    |   movel([0.123619, -1.308505, -2.621717, -0.782167, 1.570796, 1.694415],accel_mss,speed_ms,0,blend_radius_m)
    |   movel([0.123541, -1.308897, -2.621479, -0.782012, 1.570796, 1.694337],accel_mss,speed_ms,0,blend_radius_m)
    |   movel([0.123274, -1.309201, -2.621295, -0.781893, 1.570796, 1.694070],accel_mss,speed_ms,0,blend_radius_m)
    |   movel([0.122788, -1.309523, -2.621100, -0.781766, 1.570796, 1.693584],accel_mss,speed_ms,0,blend_radius_m)
    |   movel([0.122358, -1.309528, -2.621097, -0.781764, 1.570796, 1.693155],accel_mss,speed_ms,0,blend_radius_m)
    |   movel([0.122204, -1.309206, -2.621292, -0.781891, 1.570796, 1.693000],accel_mss,speed_ms,0,blend_radius_m)
    |   movel([0.122399, -1.308718, -2.621588, -0.782083, 1.570796, 1.693196],accel_mss,speed_ms,0,blend_radius_m)
    |   speed_ms = 0.003
    |   movel([0.122399, -1.294954, -2.615092, -0.802344, 1.570796, 1.693196],accel_mss,speed_ms,0,blend_radius_m)
    |   speed_ms = 1.000
    |   movel([0.122399, -1.268722, -2.601712, -0.841955, 1.570796, 1.693196],accel_mss,speed_ms,0,blend_radius_m)
    |   movel([0.122299, -1.268148, -2.602040, -0.842201, 1.570796, 1.693095],accel_mss,speed_ms,0,blend_radius_m)
    |   movel([0.122299, -1.294388, -2.615427, -0.802573, 1.570796, 1.693095],accel_mss,speed_ms,0,blend_radius_m)
    |   speed_ms = 0.003
    |   movel([0.122299, -1.304675, -2.620314, -0.787400, 1.570796, 1.693095],accel_mss,speed_ms,0,blend_radius_m)
    |   speed_ms = 0.007
    |   movel([0.123492, -1.303784, -2.620850, -0.787755, 1.570796, 1.694289],accel_mss,speed_ms,0,blend_radius_m)
    |   movel([0.124884, -1.303405, -2.621078, -0.787906, 1.570796, 1.695680],accel_mss,speed_ms,0,blend_radius_m)
    |   movel([0.125943, -1.303780, -2.620852, -0.787756, 1.570796, 1.696740],accel_mss,speed_ms,0,blend_radius_m)
    |   movel([0.126327, -1.304786, -2.620247, -0.787356, 1.570796, 1.697123],accel_mss,speed_ms,0,blend_radius_m)
    |   movel([0.125902, -1.306088, -2.619462, -0.786839, 1.570796, 1.696698],accel_mss,speed_ms,0,blend_radius_m)
    |   movel([0.125601, -1.306535, -2.619192, -0.786662, 1.570796, 1.696398],accel_mss,speed_ms,0,blend_radius_m)
    |   movel([0.125298, -1.306889, -2.618978, -0.786522, 1.570796, 1.696095],accel_mss,speed_ms,0,blend_radius_m)
    |   movel([0.124939, -1.307203, -2.618788, -0.786398, 1.570796, 1.695735],accel_mss,speed_ms,0,blend_radius_m)
    |   movel([0.124479, -1.307524, -2.618594, -0.786271, 1.570796, 1.695275],accel_mss,speed_ms,0,blend_radius_m)
    |   movel([0.123696, -1.307924, -2.618351, -0.786113, 1.570796, 1.694492],accel_mss,speed_ms,0,blend_radius_m)
    |   movel([0.122962, -1.308104, -2.618242, -0.786043, 1.570796, 1.693758],accel_mss,speed_ms,0,blend_radius_m)
    |   movel([0.122312, -1.308051, -2.618275, -0.786064, 1.570796, 1.693109],accel_mss,speed_ms,0,blend_radius_m)
    |   movel([0.121777, -1.307771, -2.618444, -0.786174, 1.570796, 1.692573],accel_mss,speed_ms,0,blend_radius_m)
    |   movel([0.121328, -1.306933, -2.618951, -0.786504, 1.570796, 1.692124],accel_mss,speed_ms,0,blend_radius_m)
    |   movel([0.121515, -1.305815, -2.619627, -0.786947, 1.570796, 1.692311],accel_mss,speed_ms,0,blend_radius_m)
    |   movel([0.122299, -1.304675, -2.620314, -0.787400, 1.570796, 1.693095],accel_mss,speed_ms,0,blend_radius_m)
    |   speed_ms = 0.003
    |   movel([0.122299, -1.308158, -2.621927, -0.782304, 1.570796, 1.693095],accel_mss,speed_ms,0,blend_radius_m)
    |   speed_ms = 0.007
    |   movel([0.123492, -1.307270, -2.622464, -0.782655, 1.570796, 1.694289],accel_mss,speed_ms,0,blend_radius_m)
    |   movel([0.124884, -1.306892, -2.622692, -0.782805, 1.570796, 1.695680],accel_mss,speed_ms,0,blend_radius_m)
    |   movel([0.125943, -1.307266, -2.622466, -0.782657, 1.570796, 1.696740],accel_mss,speed_ms,0,blend_radius_m)
    |   movel([0.126327, -1.308269, -2.621860, -0.782260, 1.570796, 1.697123],accel_mss,speed_ms,0,blend_radius_m)
    |   movel([0.125902, -1.309569, -2.621072, -0.781748, 1.570796, 1.696698],accel_mss,speed_ms,0,blend_radius_m)
    |   movel([0.125601, -1.310014, -2.620802, -0.781573, 1.570796, 1.696398],accel_mss,speed_ms,0,blend_radius_m)
    |   movel([0.125298, -1.310367, -2.620587, -0.781435, 1.570796, 1.696095],accel_mss,speed_ms,0,blend_radius_m)
    |   movel([0.124939, -1.310681, -2.620396, -0.781312, 1.570796, 1.695735],accel_mss,speed_ms,0,blend_radius_m)
    |   movel([0.124479, -1.311001, -2.620202, -0.781187, 1.570796, 1.695275],accel_mss,speed_ms,0,blend_radius_m)
    |   movel([0.123696, -1.311401, -2.619958, -0.781030, 1.570796, 1.694492],accel_mss,speed_ms,0,blend_radius_m)
    |   movel([0.122962, -1.311579, -2.619849, -0.780961, 1.570796, 1.693758],accel_mss,speed_ms,0,blend_radius_m)
    |   movel([0.122312, -1.311526, -2.619881, -0.780981, 1.570796, 1.693109],accel_mss,speed_ms,0,blend_radius_m)
    |   movel([0.121777, -1.311247, -2.620052, -0.781090, 1.570796, 1.692573],accel_mss,speed_ms,0,blend_radius_m)
    |   movel([0.121328, -1.310412, -2.620560, -0.781417, 1.570796, 1.692124],accel_mss,speed_ms,0,blend_radius_m)
    |   movel([0.121515, -1.309296, -2.621237, -0.781855, 1.570796, 1.692311],accel_mss,speed_ms,0,blend_radius_m)
    |   movel([0.122299, -1.308158, -2.621927, -0.782304, 1.570796, 1.693095],accel_mss,speed_ms,0,blend_radius_m)
    |   speed_ms = 0.003
    |   movel([0.122299, -1.294388, -2.615427, -0.802573, 1.570796, 1.693095],accel_mss,speed_ms,0,blend_radius_m)
    |   speed_ms = 1.000
    |   movel([0.122299, -1.268148, -2.602040, -0.842201, 1.570796, 1.693095],accel_mss,speed_ms,0,blend_radius_m)
    |   movel([0.122125, -1.267925, -2.602168, -0.842296, 1.570796, 1.692921],accel_mss,speed_ms,0,blend_radius_m)
    |   movel([0.122125, -1.294168, -2.615558, -0.802663, 1.570796, 1.692921],accel_mss,speed_ms,0,blend_radius_m)
    |   speed_ms = 0.003
    |   movel([0.122125, -1.304456, -2.620446, -0.787487, 1.570796, 1.692921],accel_mss,speed_ms,0,blend_radius_m)
    |   speed_ms = 0.007
    |   movel([0.122925, -1.303761, -2.620864, -0.787764, 1.570796, 1.693721],accel_mss,speed_ms,0,blend_radius_m)
    |   movel([0.123725, -1.303295, -2.621144, -0.787950, 1.570796, 1.694522],accel_mss,speed_ms,0,blend_radius_m)
    |   movel([0.124531, -1.303058, -2.621286, -0.788045, 1.570796, 1.695328],accel_mss,speed_ms,0,blend_radius_m)
    |   movel([0.125337, -1.303049, -2.621291, -0.788049, 1.570796, 1.696133],accel_mss,speed_ms,0,blend_radius_m)
    |   movel([0.125825, -1.303152, -2.621230, -0.788008, 1.570796, 1.696622],accel_mss,speed_ms,0,blend_radius_m)
    |   movel([0.126187, -1.303319, -2.621130, -0.787941, 1.570796, 1.696983],accel_mss,speed_ms,0,blend_radius_m)
    |   movel([0.126450, -1.303564, -2.620982, -0.787843, 1.570796, 1.697247],accel_mss,speed_ms,0,blend_radius_m)
    |   movel([0.126642, -1.303905, -2.620777, -0.787707, 1.570796, 1.697439],accel_mss,speed_ms,0,blend_radius_m)
    |   movel([0.126720, -1.304353, -2.620508, -0.787528, 1.570796, 1.697516],accel_mss,speed_ms,0,blend_radius_m)
    |   movel([0.126726, -1.304642, -2.620334, -0.787413, 1.570796, 1.697522],accel_mss,speed_ms,0,blend_radius_m)
    |   movel([0.126703, -1.304915, -2.620169, -0.787304, 1.570796, 1.697499],accel_mss,speed_ms,0,blend_radius_m)
    |   movel([0.126188, -1.306244, -2.619368, -0.786777, 1.570796, 1.696984],accel_mss,speed_ms,0,blend_radius_m)
    |   movel([0.125095, -1.307462, -2.618631, -0.786296, 1.570796, 1.695892],accel_mss,speed_ms,0,blend_radius_m)
    |   movel([0.123703, -1.308267, -2.618143, -0.785979, 1.570796, 1.694499],accel_mss,speed_ms,0,blend_radius_m)
    |   movel([0.122352, -1.308465, -2.618023, -0.785901, 1.570796, 1.693148],accel_mss,speed_ms,0,blend_radius_m)
    |   movel([0.121300, -1.308016, -2.618296, -0.786077, 1.570796, 1.692096],accel_mss,speed_ms,0,blend_radius_m)
    |   movel([0.120873, -1.307051, -2.618880, -0.786458, 1.570796, 1.691669],accel_mss,speed_ms,0,blend_radius_m)
    |   movel([0.121170, -1.305774, -2.619652, -0.786963, 1.570796, 1.691966],accel_mss,speed_ms,0,blend_radius_m)
    |   movel([0.122125, -1.304456, -2.620446, -0.787487, 1.570796, 1.692921],accel_mss,speed_ms,0,blend_radius_m)
    |   speed_ms = 0.003
    |   movel([0.122125, -1.307940, -2.622059, -0.782390, 1.570796, 1.692921],accel_mss,speed_ms,0,blend_radius_m)
    |   speed_ms = 0.007
    |   movel([0.122925, -1.307246, -2.622478, -0.782665, 1.570796, 1.693721],accel_mss,speed_ms,0,blend_radius_m)
    |   movel([0.123725, -1.306782, -2.622759, -0.782849, 1.570796, 1.694522],accel_mss,speed_ms,0,blend_radius_m)
    |   movel([0.124531, -1.306545, -2.622901, -0.782943, 1.570796, 1.695328],accel_mss,speed_ms,0,blend_radius_m)
    |   movel([0.125337, -1.306536, -2.622906, -0.782946, 1.570796, 1.696133],accel_mss,speed_ms,0,blend_radius_m)
    |   movel([0.125825, -1.306639, -2.622845, -0.782905, 1.570796, 1.696622],accel_mss,speed_ms,0,blend_radius_m)
    |   movel([0.126187, -1.306805, -2.622744, -0.782839, 1.570796, 1.696983],accel_mss,speed_ms,0,blend_radius_m)
    |   movel([0.126450, -1.307050, -2.622597, -0.782742, 1.570796, 1.697247],accel_mss,speed_ms,0,blend_radius_m)
    |   movel([0.126642, -1.307390, -2.622391, -0.782608, 1.570796, 1.697439],accel_mss,speed_ms,0,blend_radius_m)
    |   movel([0.126720, -1.307837, -2.622121, -0.782431, 1.570796, 1.697516],accel_mss,speed_ms,0,blend_radius_m)
    |   movel([0.126726, -1.308125, -2.621947, -0.782317, 1.570796, 1.697522],accel_mss,speed_ms,0,blend_radius_m)
    |   movel([0.126703, -1.308398, -2.621782, -0.782209, 1.570796, 1.697499],accel_mss,speed_ms,0,blend_radius_m)
    |   movel([0.126188, -1.309724, -2.620978, -0.781687, 1.570796, 1.696984],accel_mss,speed_ms,0,blend_radius_m)
    |   movel([0.125095, -1.310939, -2.620239, -0.781211, 1.570796, 1.695892],accel_mss,speed_ms,0,blend_radius_m)
    |   movel([0.123703, -1.311742, -2.619750, -0.780897, 1.570796, 1.694499],accel_mss,speed_ms,0,blend_radius_m)
    |   movel([0.122352, -1.311940, -2.619629, -0.780820, 1.570796, 1.693148],accel_mss,speed_ms,0,blend_radius_m)
    |   movel([0.121300, -1.311492, -2.619902, -0.780995, 1.570796, 1.692096],accel_mss,speed_ms,0,blend_radius_m)
    |   movel([0.120873, -1.310529, -2.620488, -0.781371, 1.570796, 1.691669],accel_mss,speed_ms,0,blend_radius_m)
    |   movel([0.121170, -1.309255, -2.621262, -0.781871, 1.570796, 1.691966],accel_mss,speed_ms,0,blend_radius_m)
    |   movel([0.122125, -1.307940, -2.622059, -0.782390, 1.570796, 1.692921],accel_mss,speed_ms,0,blend_radius_m)
    |   speed_ms = 0.003
    |   movel([0.122125, -1.294168, -2.615558, -0.802663, 1.570796, 1.692921],accel_mss,speed_ms,0,blend_radius_m)
    |   speed_ms = 1.000
    |   movel([0.122125, -1.267925, -2.602168, -0.842296, 1.570796, 1.692921],accel_mss,speed_ms,0,blend_radius_m)
    |   movel([0.121075, -1.274686, -2.598277, -0.839426, 1.570796, 1.691871],accel_mss,speed_ms,0,blend_radius_m)
    |   movel([0.121075, -1.300833, -2.611578, -0.799978, 1.570796, 1.691871],accel_mss,speed_ms,0,blend_radius_m)
    |   speed_ms = 0.003
    |   movel([0.121075, -1.311078, -2.616433, -0.784878, 1.570796, 1.691871],accel_mss,speed_ms,0,blend_radius_m)
    |   speed_ms = 0.007
    |   movel([0.123533, -1.310110, -2.617023, -0.785256, 1.570796, 1.694329],accel_mss,speed_ms,0,blend_radius_m)
    |   movel([0.125640, -1.309106, -2.617634, -0.785649, 1.570796, 1.696436],accel_mss,speed_ms,0,blend_radius_m)
    |   movel([0.127292, -1.308097, -2.618247, -0.786046, 1.570796, 1.698089],accel_mss,speed_ms,0,blend_radius_m)
    |   movel([0.127580, -1.307905, -2.618363, -0.786121, 1.570796, 1.698376],accel_mss,speed_ms,0,blend_radius_m)
    |   movel([0.127853, -1.307745, -2.618460, -0.786184, 1.570796, 1.698649],accel_mss,speed_ms,0,blend_radius_m)
    |   movel([0.128201, -1.307606, -2.618544, -0.786239, 1.570796, 1.698997],accel_mss,speed_ms,0,blend_radius_m)
    |   movel([0.128478, -1.307907, -2.618362, -0.786121, 1.570796, 1.699274],accel_mss,speed_ms,0,blend_radius_m)
    |   movel([0.128527, -1.308214, -2.618176, -0.786000, 1.570796, 1.699324],accel_mss,speed_ms,0,blend_radius_m)
    |   movel([0.128494, -1.308549, -2.617972, -0.785868, 1.570796, 1.699291],accel_mss,speed_ms,0,blend_radius_m)
    |   movel([0.128245, -1.308983, -2.617708, -0.785697, 1.570796, 1.699041],accel_mss,speed_ms,0,blend_radius_m)
    |   movel([0.127949, -1.309233, -2.617557, -0.785599, 1.570796, 1.698745],accel_mss,speed_ms,0,blend_radius_m)
    |   movel([0.127334, -1.309676, -2.617287, -0.785426, 1.570796, 1.698131],accel_mss,speed_ms,0,blend_radius_m)
    |   movel([0.126550, -1.310204, -2.616966, -0.785219, 1.570796, 1.697346],accel_mss,speed_ms,0,blend_radius_m)
    |   movel([0.126053, -1.310466, -2.616806, -0.785117, 1.570796, 1.696849],accel_mss,speed_ms,0,blend_radius_m)
    |   movel([0.125676, -1.310561, -2.616748, -0.785080, 1.570796, 1.696472],accel_mss,speed_ms,0,blend_radius_m)
    |   movel([0.125323, -1.310521, -2.616772, -0.785095, 1.570796, 1.696119],accel_mss,speed_ms,0,blend_radius_m)
    |   movel([0.125032, -1.310484, -2.616795, -0.785110, 1.570796, 1.695828],accel_mss,speed_ms,0,blend_radius_m)
    |   movel([0.124704, -1.310732, -2.616644, -0.785013, 1.570796, 1.695500],accel_mss,speed_ms,0,blend_radius_m)
    |   movel([0.124538, -1.311064, -2.616441, -0.784884, 1.570796, 1.695334],accel_mss,speed_ms,0,blend_radius_m)
    |   movel([0.124342, -1.311404, -2.616233, -0.784751, 1.570796, 1.695138],accel_mss,speed_ms,0,blend_radius_m)
    |   movel([0.123812, -1.311686, -2.616061, -0.784642, 1.570796, 1.694608],accel_mss,speed_ms,0,blend_radius_m)
    |   movel([0.123019, -1.311995, -2.615873, -0.784522, 1.570796, 1.693815],accel_mss,speed_ms,0,blend_radius_m)
    |   movel([0.122341, -1.312263, -2.615709, -0.784418, 1.570796, 1.693137],accel_mss,speed_ms,0,blend_radius_m)
    |   movel([0.121606, -1.312553, -2.615531, -0.784305, 1.570796, 1.692402],accel_mss,speed_ms,0,blend_radius_m)
    |   movel([0.119881, -1.313195, -2.615138, -0.784056, 1.570796, 1.690677],accel_mss,speed_ms,0,blend_radius_m)
    |   movel([0.118261, -1.313723, -2.614814, -0.783852, 1.570796, 1.689057],accel_mss,speed_ms,0,blend_radius_m)
    |   movel([0.116698, -1.314145, -2.614554, -0.783689, 1.570796, 1.687494],accel_mss,speed_ms,0,blend_radius_m)
    |   movel([0.115130, -1.314485, -2.614345, -0.783558, 1.570796, 1.685926],accel_mss,speed_ms,0,blend_radius_m)
    |   movel([0.114283, -1.314653, -2.614242, -0.783494, 1.570796, 1.685079],accel_mss,speed_ms,0,blend_radius_m)
    |   movel([0.113758, -1.314782, -2.614163, -0.783444, 1.570796, 1.684554],accel_mss,speed_ms,0,blend_radius_m)
    |   movel([0.113408, -1.314897, -2.614092, -0.783400, 1.570796, 1.684204],accel_mss,speed_ms,0,blend_radius_m)
    |   movel([0.113047, -1.315126, -2.613951, -0.783312, 1.570796, 1.683843],accel_mss,speed_ms,0,blend_radius_m)
    |   movel([0.112717, -1.315125, -2.613952, -0.783312, 1.570796, 1.683513],accel_mss,speed_ms,0,blend_radius_m)
    |   movel([0.112491, -1.315087, -2.613975, -0.783327, 1.570796, 1.683287],accel_mss,speed_ms,0,blend_radius_m)
    |   movel([0.112110, -1.315203, -2.613904, -0.783282, 1.570796, 1.682907],accel_mss,speed_ms,0,blend_radius_m)
    |   movel([0.111865, -1.315072, -2.613984, -0.783332, 1.570796, 1.682661],accel_mss,speed_ms,0,blend_radius_m)
    |   movel([0.111544, -1.314898, -2.614091, -0.783399, 1.570796, 1.682340],accel_mss,speed_ms,0,blend_radius_m)
    |   movel([0.111224, -1.314841, -2.614126, -0.783421, 1.570796, 1.682020],accel_mss,speed_ms,0,blend_radius_m)
    |   movel([0.110794, -1.314811, -2.614145, -0.783433, 1.570796, 1.681590],accel_mss,speed_ms,0,blend_radius_m)
    |   movel([0.109970, -1.314754, -2.614180, -0.783455, 1.570796, 1.680766],accel_mss,speed_ms,0,blend_radius_m)
    |   movel([0.109663, -1.314650, -2.614244, -0.783495, 1.570796, 1.680459],accel_mss,speed_ms,0,blend_radius_m)
    |   movel([0.109585, -1.314439, -2.614374, -0.783576, 1.570796, 1.680381],accel_mss,speed_ms,0,blend_radius_m)
    |   movel([0.109700, -1.314035, -2.614622, -0.783732, 1.570796, 1.680497],accel_mss,speed_ms,0,blend_radius_m)
    |   movel([0.109948, -1.313528, -2.614934, -0.783928, 1.570796, 1.680744],accel_mss,speed_ms,0,blend_radius_m)
    |   movel([0.110182, -1.313278, -2.615087, -0.784024, 1.570796, 1.680979],accel_mss,speed_ms,0,blend_radius_m)
    |   movel([0.110476, -1.313177, -2.615149, -0.784063, 1.570796, 1.681272],accel_mss,speed_ms,0,blend_radius_m)
    |   movel([0.110954, -1.313204, -2.615132, -0.784053, 1.570796, 1.681750],accel_mss,speed_ms,0,blend_radius_m)
    |   movel([0.112252, -1.313249, -2.615105, -0.784036, 1.570796, 1.683048],accel_mss,speed_ms,0,blend_radius_m)
    |   movel([0.113926, -1.313054, -2.615224, -0.784111, 1.570796, 1.684722],accel_mss,speed_ms,0,blend_radius_m)
    |   movel([0.115954, -1.312630, -2.615484, -0.784275, 1.570796, 1.686750],accel_mss,speed_ms,0,blend_radius_m)
    |   movel([0.118344, -1.311973, -2.615886, -0.784530, 1.570796, 1.689140],accel_mss,speed_ms,0,blend_radius_m)
    |   movel([0.121075, -1.311078, -2.616433, -0.784878, 1.570796, 1.691871],accel_mss,speed_ms,0,blend_radius_m)
    |   speed_ms = 0.003
    |   movel([0.121075, -1.314547, -2.618034, -0.779808, 1.570796, 1.691871],accel_mss,speed_ms,0,blend_radius_m)
    |   speed_ms = 0.007
    |   movel([0.123533, -1.313581, -2.618626, -0.780182, 1.570796, 1.694329],accel_mss,speed_ms,0,blend_radius_m)
    |   movel([0.125640, -1.312579, -2.619239, -0.780571, 1.570796, 1.696436],accel_mss,speed_ms,0,blend_radius_m)
    |   movel([0.127292, -1.311572, -2.619853, -0.780963, 1.570796, 1.698089],accel_mss,speed_ms,0,blend_radius_m)
    |   movel([0.127580, -1.311381, -2.619970, -0.781038, 1.570796, 1.698376],accel_mss,speed_ms,0,blend_radius_m)
    |   movel([0.127853, -1.311222, -2.620067, -0.781100, 1.570796, 1.698649],accel_mss,speed_ms,0,blend_radius_m)
    |   movel([0.128201, -1.311082, -2.620152, -0.781155, 1.570796, 1.698997],accel_mss,speed_ms,0,blend_radius_m)
    |   movel([0.128478, -1.311383, -2.619969, -0.781037, 1.570796, 1.699274],accel_mss,speed_ms,0,blend_radius_m)
    |   movel([0.128527, -1.311689, -2.619782, -0.780918, 1.570796, 1.699324],accel_mss,speed_ms,0,blend_radius_m)
    |   movel([0.128494, -1.312024, -2.619578, -0.780787, 1.570796, 1.699291],accel_mss,speed_ms,0,blend_radius_m)
    |   movel([0.128245, -1.312457, -2.619313, -0.780618, 1.570796, 1.699041],accel_mss,speed_ms,0,blend_radius_m)
    |   movel([0.127949, -1.312706, -2.619161, -0.780521, 1.570796, 1.698745],accel_mss,speed_ms,0,blend_radius_m)
    |   movel([0.127334, -1.313148, -2.618891, -0.780350, 1.570796, 1.698131],accel_mss,speed_ms,0,blend_radius_m)
    |   movel([0.126550, -1.313675, -2.618569, -0.780145, 1.570796, 1.697346],accel_mss,speed_ms,0,blend_radius_m)
    |   movel([0.126053, -1.313937, -2.618408, -0.780044, 1.570796, 1.696849],accel_mss,speed_ms,0,blend_radius_m)
    |   movel([0.125676, -1.314031, -2.618351, -0.780007, 1.570796, 1.696472],accel_mss,speed_ms,0,blend_radius_m)
    |   movel([0.125323, -1.313991, -2.618375, -0.780023, 1.570796, 1.696119],accel_mss,speed_ms,0,blend_radius_m)
    |   movel([0.125032, -1.313954, -2.618398, -0.780037, 1.570796, 1.695828],accel_mss,speed_ms,0,blend_radius_m)
    |   movel([0.124704, -1.314201, -2.618246, -0.779941, 1.570796, 1.695500],accel_mss,speed_ms,0,blend_radius_m)
    |   movel([0.124538, -1.314533, -2.618043, -0.779813, 1.570796, 1.695334],accel_mss,speed_ms,0,blend_radius_m)
    |   movel([0.124342, -1.314872, -2.617834, -0.779682, 1.570796, 1.695138],accel_mss,speed_ms,0,blend_radius_m)
    |   movel([0.123812, -1.315153, -2.617662, -0.779574, 1.570796, 1.694608],accel_mss,speed_ms,0,blend_radius_m)
    |   movel([0.123019, -1.315461, -2.617473, -0.779455, 1.570796, 1.693815],accel_mss,speed_ms,0,blend_radius_m)
    |   movel([0.122341, -1.315729, -2.617308, -0.779352, 1.570796, 1.693137],accel_mss,speed_ms,0,blend_radius_m)
    |   movel([0.121606, -1.316018, -2.617130, -0.779241, 1.570796, 1.692402],accel_mss,speed_ms,0,blend_radius_m)
    |   movel([0.119881, -1.316659, -2.616736, -0.778994, 1.570796, 1.690677],accel_mss,speed_ms,0,blend_radius_m)
    |   movel([0.118261, -1.317185, -2.616411, -0.778793, 1.570796, 1.689057],accel_mss,speed_ms,0,blend_radius_m)
    |   movel([0.116698, -1.317607, -2.616151, -0.778631, 1.570796, 1.687494],accel_mss,speed_ms,0,blend_radius_m)
    |   movel([0.115130, -1.317946, -2.615941, -0.778502, 1.570796, 1.685926],accel_mss,speed_ms,0,blend_radius_m)
    |   movel([0.114283, -1.318114, -2.615838, -0.778438, 1.570796, 1.685079],accel_mss,speed_ms,0,blend_radius_m)
    |   movel([0.113758, -1.318242, -2.615758, -0.778389, 1.570796, 1.684554],accel_mss,speed_ms,0,blend_radius_m)
    |   movel([0.113408, -1.318357, -2.615687, -0.778345, 1.570796, 1.684204],accel_mss,speed_ms,0,blend_radius_m)
    |   movel([0.113047, -1.318585, -2.615546, -0.778258, 1.570796, 1.683843],accel_mss,speed_ms,0,blend_radius_m)
    |   movel([0.112717, -1.318584, -2.615547, -0.778258, 1.570796, 1.683513],accel_mss,speed_ms,0,blend_radius_m)
    |   movel([0.112491, -1.318547, -2.615570, -0.778273, 1.570796, 1.683287],accel_mss,speed_ms,0,blend_radius_m)
    |   movel([0.112110, -1.318662, -2.615498, -0.778229, 1.570796, 1.682907],accel_mss,speed_ms,0,blend_radius_m)
    |   movel([0.111865, -1.318532, -2.615579, -0.778278, 1.570796, 1.682661],accel_mss,speed_ms,0,blend_radius_m)
    |   movel([0.111544, -1.318358, -2.615686, -0.778344, 1.570796, 1.682340],accel_mss,speed_ms,0,blend_radius_m)
    |   movel([0.111224, -1.318301, -2.615722, -0.778366, 1.570796, 1.682020],accel_mss,speed_ms,0,blend_radius_m)
    |   movel([0.110794, -1.318271, -2.615740, -0.778378, 1.570796, 1.681590],accel_mss,speed_ms,0,blend_radius_m)
    |   movel([0.109970, -1.318214, -2.615775, -0.778399, 1.570796, 1.680766],accel_mss,speed_ms,0,blend_radius_m)
    |   movel([0.109663, -1.318110, -2.615840, -0.778439, 1.570796, 1.680459],accel_mss,speed_ms,0,blend_radius_m)
    |   movel([0.109585, -1.317900, -2.615970, -0.778519, 1.570796, 1.680381],accel_mss,speed_ms,0,blend_radius_m)
    |   movel([0.109700, -1.317497, -2.616219, -0.778673, 1.570796, 1.680497],accel_mss,speed_ms,0,blend_radius_m)
    |   movel([0.109948, -1.316991, -2.616531, -0.778867, 1.570796, 1.680744],accel_mss,speed_ms,0,blend_radius_m)
    |   movel([0.110182, -1.316742, -2.616684, -0.778963, 1.570796, 1.680979],accel_mss,speed_ms,0,blend_radius_m)
    |   movel([0.110476, -1.316641, -2.616747, -0.779001, 1.570796, 1.681272],accel_mss,speed_ms,0,blend_radius_m)
    |   movel([0.110954, -1.316668, -2.616730, -0.778991, 1.570796, 1.681750],accel_mss,speed_ms,0,blend_radius_m)
    |   movel([0.112252, -1.316712, -2.616703, -0.778974, 1.570796, 1.683048],accel_mss,speed_ms,0,blend_radius_m)
    |   movel([0.113926, -1.316518, -2.616822, -0.779048, 1.570796, 1.684722],accel_mss,speed_ms,0,blend_radius_m)
    |   movel([0.115954, -1.316095, -2.617083, -0.779211, 1.570796, 1.686750],accel_mss,speed_ms,0,blend_radius_m)
    |   movel([0.118344, -1.315440, -2.617486, -0.779463, 1.570796, 1.689140],accel_mss,speed_ms,0,blend_radius_m)
    |   movel([0.121075, -1.314547, -2.618034, -0.779808, 1.570796, 1.691871],accel_mss,speed_ms,0,blend_radius_m)
    |   speed_ms = 0.003
    |   movel([0.121075, -1.300833, -2.611578, -0.799978, 1.570796, 1.691871],accel_mss,speed_ms,0,blend_radius_m)
    |   speed_ms = 1.000
    |   movel([0.121075, -1.274686, -2.598277, -0.839426, 1.570796, 1.691871],accel_mss,speed_ms,0,blend_radius_m)
    |   movel([0.121859, -1.276472, -2.597239, -0.838677, 1.570796, 1.692655],accel_mss,speed_ms,0,blend_radius_m)
    |   movel([0.121859, -1.302594, -2.610517, -0.799278, 1.570796, 1.692655],accel_mss,speed_ms,0,blend_radius_m)
    |   speed_ms = 0.003
    |   movel([0.121859, -1.312827, -2.615363, -0.784199, 1.570796, 1.692655],accel_mss,speed_ms,0,blend_radius_m)
    |   speed_ms = 0.007
    |   movel([0.122991, -1.312380, -2.615637, -0.784372, 1.570796, 1.693788],accel_mss,speed_ms,0,blend_radius_m)
    |   movel([0.123440, -1.312231, -2.615728, -0.784430, 1.570796, 1.694237],accel_mss,speed_ms,0,blend_radius_m)
    |   movel([0.123730, -1.312196, -2.615749, -0.784443, 1.570796, 1.694527],accel_mss,speed_ms,0,blend_radius_m)
    |   movel([0.124033, -1.312239, -2.615723, -0.784427, 1.570796, 1.694829],accel_mss,speed_ms,0,blend_radius_m)
    |   movel([0.124294, -1.312303, -2.615684, -0.784402, 1.570796, 1.695090],accel_mss,speed_ms,0,blend_radius_m)
    |   movel([0.124688, -1.312083, -2.615819, -0.784487, 1.570796, 1.695484],accel_mss,speed_ms,0,blend_radius_m)
    |   movel([0.124878, -1.311816, -2.615982, -0.784591, 1.570796, 1.695675],accel_mss,speed_ms,0,blend_radius_m)
    |   movel([0.125008, -1.311555, -2.616141, -0.784692, 1.570796, 1.695805],accel_mss,speed_ms,0,blend_radius_m)
    |   movel([0.125321, -1.311234, -2.616338, -0.784818, 1.570796, 1.696117],accel_mss,speed_ms,0,blend_radius_m)
    |   movel([0.125785, -1.311040, -2.616456, -0.784893, 1.570796, 1.696581],accel_mss,speed_ms,0,blend_radius_m)
    |   movel([0.126205, -1.310800, -2.616602, -0.784987, 1.570796, 1.697002],accel_mss,speed_ms,0,blend_radius_m)
    |   movel([0.126690, -1.310497, -2.616787, -0.785105, 1.570796, 1.697486],accel_mss,speed_ms,0,blend_radius_m)
    |   movel([0.127180, -1.310170, -2.616987, -0.785233, 1.570796, 1.697977],accel_mss,speed_ms,0,blend_radius_m)
    |   movel([0.127663, -1.309845, -2.617185, -0.785360, 1.570796, 1.698460],accel_mss,speed_ms,0,blend_radius_m)
    |   movel([0.128093, -1.309581, -2.617345, -0.785463, 1.570796, 1.698890],accel_mss,speed_ms,0,blend_radius_m)
    |   movel([0.128444, -1.309388, -2.617462, -0.785539, 1.570796, 1.699240],accel_mss,speed_ms,0,blend_radius_m)
    |   movel([0.128700, -1.309411, -2.617449, -0.785530, 1.570796, 1.699496],accel_mss,speed_ms,0,blend_radius_m)
    |   movel([0.128790, -1.309863, -2.617173, -0.785353, 1.570796, 1.699587],accel_mss,speed_ms,0,blend_radius_m)
    |   movel([0.128773, -1.310342, -2.616881, -0.785165, 1.570796, 1.699569],accel_mss,speed_ms,0,blend_radius_m)
    |   movel([0.128639, -1.310639, -2.616700, -0.785049, 1.570796, 1.699436],accel_mss,speed_ms,0,blend_radius_m)
    |   movel([0.128342, -1.311007, -2.616476, -0.784906, 1.570796, 1.699139],accel_mss,speed_ms,0,blend_radius_m)
    |   movel([0.127842, -1.311459, -2.616200, -0.784730, 1.570796, 1.698638],accel_mss,speed_ms,0,blend_radius_m)
    |   movel([0.127119, -1.312016, -2.615860, -0.784513, 1.570796, 1.697915],accel_mss,speed_ms,0,blend_radius_m)
    |   movel([0.126316, -1.312577, -2.615516, -0.784296, 1.570796, 1.697112],accel_mss,speed_ms,0,blend_radius_m)
    |   movel([0.125554, -1.313058, -2.615222, -0.784110, 1.570796, 1.696350],accel_mss,speed_ms,0,blend_radius_m)
    |   movel([0.123821, -1.314003, -2.614641, -0.783744, 1.570796, 1.694617],accel_mss,speed_ms,0,blend_radius_m)
    |   movel([0.122103, -1.314798, -2.614153, -0.783438, 1.570796, 1.692899],accel_mss,speed_ms,0,blend_radius_m)
    |   movel([0.120238, -1.315511, -2.613714, -0.783164, 1.570796, 1.691034],accel_mss,speed_ms,0,blend_radius_m)
    |   movel([0.118050, -1.316214, -2.613280, -0.782894, 1.570796, 1.688847],accel_mss,speed_ms,0,blend_radius_m)
    |   movel([0.115606, -1.316871, -2.612875, -0.782643, 1.570796, 1.686403],accel_mss,speed_ms,0,blend_radius_m)
    |   movel([0.113590, -1.317254, -2.612638, -0.782497, 1.570796, 1.684386],accel_mss,speed_ms,0,blend_radius_m)
    |   movel([0.111851, -1.317389, -2.612554, -0.782446, 1.570796, 1.682647],accel_mss,speed_ms,0,blend_radius_m)
    |   movel([0.110255, -1.317292, -2.612614, -0.782482, 1.570796, 1.681051],accel_mss,speed_ms,0,blend_radius_m)
    |   movel([0.109457, -1.317140, -2.612708, -0.782540, 1.570796, 1.680254],accel_mss,speed_ms,0,blend_radius_m)
    |   movel([0.109068, -1.316938, -2.612833, -0.782618, 1.570796, 1.679864],accel_mss,speed_ms,0,blend_radius_m)
    |   movel([0.108931, -1.316617, -2.613032, -0.782740, 1.570796, 1.679727],accel_mss,speed_ms,0,blend_radius_m)
    |   movel([0.108994, -1.316104, -2.613349, -0.782937, 1.570796, 1.679791],accel_mss,speed_ms,0,blend_radius_m)
    |   movel([0.109160, -1.315584, -2.613669, -0.783136, 1.570796, 1.679956],accel_mss,speed_ms,0,blend_radius_m)
    |   movel([0.109607, -1.315229, -2.613888, -0.783272, 1.570796, 1.680403],accel_mss,speed_ms,0,blend_radius_m)
    |   movel([0.110127, -1.315201, -2.613905, -0.783283, 1.570796, 1.680923],accel_mss,speed_ms,0,blend_radius_m)
    |   movel([0.110747, -1.315224, -2.613891, -0.783274, 1.570796, 1.681544],accel_mss,speed_ms,0,blend_radius_m)
    |   movel([0.111099, -1.315298, -2.613845, -0.783246, 1.570796, 1.681895],accel_mss,speed_ms,0,blend_radius_m)
    |   movel([0.111289, -1.315438, -2.613759, -0.783192, 1.570796, 1.682085],accel_mss,speed_ms,0,blend_radius_m)
    |   movel([0.111376, -1.315672, -2.613615, -0.783102, 1.570796, 1.682173],accel_mss,speed_ms,0,blend_radius_m)
    |   movel([0.111519, -1.315939, -2.613450, -0.783000, 1.570796, 1.682315],accel_mss,speed_ms,0,blend_radius_m)
    |   movel([0.112017, -1.316002, -2.613411, -0.782976, 1.570796, 1.682813],accel_mss,speed_ms,0,blend_radius_m)
    |   movel([0.112431, -1.315982, -2.613424, -0.782983, 1.570796, 1.683228],accel_mss,speed_ms,0,blend_radius_m)
    |   movel([0.112913, -1.315767, -2.613556, -0.783066, 1.570796, 1.683709],accel_mss,speed_ms,0,blend_radius_m)
    |   movel([0.113257, -1.315447, -2.613754, -0.783189, 1.570796, 1.684053],accel_mss,speed_ms,0,blend_radius_m)
    |   movel([0.113713, -1.315150, -2.613936, -0.783303, 1.570796, 1.684509],accel_mss,speed_ms,0,blend_radius_m)
    |   movel([0.114070, -1.315058, -2.613993, -0.783338, 1.570796, 1.684866],accel_mss,speed_ms,0,blend_radius_m)
    |   movel([0.114914, -1.314907, -2.614086, -0.783396, 1.570796, 1.685710],accel_mss,speed_ms,0,blend_radius_m)
    |   movel([0.116379, -1.314593, -2.614279, -0.783517, 1.570796, 1.687175],accel_mss,speed_ms,0,blend_radius_m)
    |   movel([0.118199, -1.314090, -2.614588, -0.783711, 1.570796, 1.688995],accel_mss,speed_ms,0,blend_radius_m)
    |   movel([0.120107, -1.313476, -2.614965, -0.783948, 1.570796, 1.690904],accel_mss,speed_ms,0,blend_radius_m)
    |   movel([0.121859, -1.312827, -2.615363, -0.784199, 1.570796, 1.692655],accel_mss,speed_ms,0,blend_radius_m)
    |   speed_ms = 0.003
    |   movel([0.121859, -1.316291, -2.616962, -0.779136, 1.570796, 1.692655],accel_mss,speed_ms,0,blend_radius_m)
    |   speed_ms = 0.007
    |   movel([0.122991, -1.315846, -2.617236, -0.779307, 1.570796, 1.693788],accel_mss,speed_ms,0,blend_radius_m)
    |   movel([0.123440, -1.315697, -2.617328, -0.779364, 1.570796, 1.694237],accel_mss,speed_ms,0,blend_radius_m)
    |   movel([0.123730, -1.315663, -2.617349, -0.779377, 1.570796, 1.694527],accel_mss,speed_ms,0,blend_radius_m)
    |   movel([0.124033, -1.315705, -2.617323, -0.779361, 1.570796, 1.694829],accel_mss,speed_ms,0,blend_radius_m)
    |   movel([0.124294, -1.315769, -2.617283, -0.779336, 1.570796, 1.695090],accel_mss,speed_ms,0,blend_radius_m)
    |   movel([0.124688, -1.315550, -2.617418, -0.779421, 1.570796, 1.695484],accel_mss,speed_ms,0,blend_radius_m)
    |   movel([0.124878, -1.315283, -2.617582, -0.779524, 1.570796, 1.695675],accel_mss,speed_ms,0,blend_radius_m)
    |   movel([0.125008, -1.315023, -2.617742, -0.779624, 1.570796, 1.695805],accel_mss,speed_ms,0,blend_radius_m)
    |   movel([0.125321, -1.314702, -2.617939, -0.779748, 1.570796, 1.696117],accel_mss,speed_ms,0,blend_radius_m)
    |   movel([0.125785, -1.314508, -2.618058, -0.779823, 1.570796, 1.696581],accel_mss,speed_ms,0,blend_radius_m)
    |   movel([0.126205, -1.314269, -2.618205, -0.779915, 1.570796, 1.697002],accel_mss,speed_ms,0,blend_radius_m)
    |   movel([0.126690, -1.313967, -2.618390, -0.780032, 1.570796, 1.697486],accel_mss,speed_ms,0,blend_radius_m)
    |   movel([0.127180, -1.313641, -2.618590, -0.780159, 1.570796, 1.697977],accel_mss,speed_ms,0,blend_radius_m)
    |   movel([0.127663, -1.313316, -2.618788, -0.780284, 1.570796, 1.698460],accel_mss,speed_ms,0,blend_radius_m)
    |   movel([0.128093, -1.313054, -2.618949, -0.780386, 1.570796, 1.698890],accel_mss,speed_ms,0,blend_radius_m)
    |   movel([0.128444, -1.312861, -2.619067, -0.780461, 1.570796, 1.699240],accel_mss,speed_ms,0,blend_radius_m)
    |   movel([0.128700, -1.312883, -2.619053, -0.780453, 1.570796, 1.699496],accel_mss,speed_ms,0,blend_radius_m)
    |   movel([0.128790, -1.313335, -2.618777, -0.780277, 1.570796, 1.699587],accel_mss,speed_ms,0,blend_radius_m)
    |   movel([0.128773, -1.313813, -2.618484, -0.780092, 1.570796, 1.699569],accel_mss,speed_ms,0,blend_radius_m)
    |   movel([0.128639, -1.314109, -2.618303, -0.779977, 1.570796, 1.699436],accel_mss,speed_ms,0,blend_radius_m)
    |   movel([0.128342, -1.314476, -2.618078, -0.779835, 1.570796, 1.699139],accel_mss,speed_ms,0,blend_radius_m)
    |   movel([0.127842, -1.314927, -2.617801, -0.779661, 1.570796, 1.698638],accel_mss,speed_ms,0,blend_radius_m)
    |   movel([0.127119, -1.315482, -2.617460, -0.779447, 1.570796, 1.697915],accel_mss,speed_ms,0,blend_radius_m)
    |   movel([0.126316, -1.316043, -2.617115, -0.779231, 1.570796, 1.697112],accel_mss,speed_ms,0,blend_radius_m)
    |   movel([0.125554, -1.316522, -2.616820, -0.779047, 1.570796, 1.696350],accel_mss,speed_ms,0,blend_radius_m)
    |   movel([0.123821, -1.317465, -2.616238, -0.778685, 1.570796, 1.694617],accel_mss,speed_ms,0,blend_radius_m)
    |   movel([0.122103, -1.318258, -2.615748, -0.778383, 1.570796, 1.692899],accel_mss,speed_ms,0,blend_radius_m)
    |   movel([0.120238, -1.318970, -2.615308, -0.778111, 1.570796, 1.691034],accel_mss,speed_ms,0,blend_radius_m)
    |   movel([0.118050, -1.319671, -2.614873, -0.777845, 1.570796, 1.688847],accel_mss,speed_ms,0,blend_radius_m)
    |   movel([0.115606, -1.320326, -2.614466, -0.777596, 1.570796, 1.686403],accel_mss,speed_ms,0,blend_radius_m)
    |   movel([0.113590, -1.320708, -2.614229, -0.777452, 1.570796, 1.684386],accel_mss,speed_ms,0,blend_radius_m)
    |   movel([0.111851, -1.320843, -2.614145, -0.777401, 1.570796, 1.682647],accel_mss,speed_ms,0,blend_radius_m)
    |   movel([0.110255, -1.320747, -2.614205, -0.777437, 1.570796, 1.681051],accel_mss,speed_ms,0,blend_radius_m)
    |   movel([0.109457, -1.320595, -2.614299, -0.777495, 1.570796, 1.680254],accel_mss,speed_ms,0,blend_radius_m)
    |   movel([0.109068, -1.320393, -2.614425, -0.777571, 1.570796, 1.679864],accel_mss,speed_ms,0,blend_radius_m)
    |   movel([0.108931, -1.320073, -2.614624, -0.777692, 1.570796, 1.679727],accel_mss,speed_ms,0,blend_radius_m)
    |   movel([0.108994, -1.319561, -2.614942, -0.777887, 1.570796, 1.679791],accel_mss,speed_ms,0,blend_radius_m)
    |   movel([0.109160, -1.319042, -2.615263, -0.778084, 1.570796, 1.679956],accel_mss,speed_ms,0,blend_radius_m)
    |   movel([0.109607, -1.318688, -2.615482, -0.778219, 1.570796, 1.680403],accel_mss,speed_ms,0,blend_radius_m)
    |   movel([0.110127, -1.318660, -2.615499, -0.778229, 1.570796, 1.680923],accel_mss,speed_ms,0,blend_radius_m)
    |   movel([0.110747, -1.318683, -2.615486, -0.778221, 1.570796, 1.681544],accel_mss,speed_ms,0,blend_radius_m)
    |   movel([0.111099, -1.318757, -2.615439, -0.778192, 1.570796, 1.681895],accel_mss,speed_ms,0,blend_radius_m)
    |   movel([0.111289, -1.318897, -2.615353, -0.778139, 1.570796, 1.682085],accel_mss,speed_ms,0,blend_radius_m)
    |   movel([0.111376, -1.319130, -2.615209, -0.778050, 1.570796, 1.682173],accel_mss,speed_ms,0,blend_radius_m)
    |   movel([0.111519, -1.319396, -2.615043, -0.777949, 1.570796, 1.682315],accel_mss,speed_ms,0,blend_radius_m)
    |   movel([0.112017, -1.319459, -2.615005, -0.777925, 1.570796, 1.682813],accel_mss,speed_ms,0,blend_radius_m)
    |   movel([0.112431, -1.319439, -2.615017, -0.777933, 1.570796, 1.683228],accel_mss,speed_ms,0,blend_radius_m)
    |   movel([0.112913, -1.319225, -2.615150, -0.778014, 1.570796, 1.683709],accel_mss,speed_ms,0,blend_radius_m)
    |   movel([0.113257, -1.318905, -2.615348, -0.778136, 1.570796, 1.684053],accel_mss,speed_ms,0,blend_radius_m)
    |   movel([0.113713, -1.318609, -2.615531, -0.778249, 1.570796, 1.684509],accel_mss,speed_ms,0,blend_radius_m)
    |   movel([0.114070, -1.318518, -2.615588, -0.778283, 1.570796, 1.684866],accel_mss,speed_ms,0,blend_radius_m)
    |   movel([0.114914, -1.318367, -2.615681, -0.778341, 1.570796, 1.685710],accel_mss,speed_ms,0,blend_radius_m)
    |   movel([0.116379, -1.318054, -2.615874, -0.778460, 1.570796, 1.687175],accel_mss,speed_ms,0,blend_radius_m)
    |   movel([0.118199, -1.317551, -2.616185, -0.778653, 1.570796, 1.688995],accel_mss,speed_ms,0,blend_radius_m)
    |   movel([0.120107, -1.316940, -2.616562, -0.778887, 1.570796, 1.690904],accel_mss,speed_ms,0,blend_radius_m)
    |   movel([0.121859, -1.316291, -2.616962, -0.779136, 1.570796, 1.692655],accel_mss,speed_ms,0,blend_radius_m)
    |   speed_ms = 0.003
    |   movel([0.121859, -1.302594, -2.610517, -0.799278, 1.570796, 1.692655],accel_mss,speed_ms,0,blend_radius_m)
    |   speed_ms = 1.000
    |   movel([0.121859, -1.276472, -2.597239, -0.838677, 1.570796, 1.692655],accel_mss,speed_ms,0,blend_radius_m)
    |   movel([0.121968, -1.273957, -2.598699, -0.839733, 1.570796, 1.692765],accel_mss,speed_ms,0,blend_radius_m)
    |   movel([0.121968, -1.300115, -2.612010, -0.800264, 1.570796, 1.692765],accel_mss,speed_ms,0,blend_radius_m)
    |   speed_ms = 0.003
    |   movel([0.121968, -1.310364, -2.616868, -0.785157, 1.570796, 1.692765],accel_mss,speed_ms,0,blend_radius_m)
    |   speed_ms = 0.007
    |   movel([0.123908, -1.309562, -2.617356, -0.785470, 1.570796, 1.694704],accel_mss,speed_ms,0,blend_radius_m)
    |   movel([0.125557, -1.308732, -2.617861, -0.785796, 1.570796, 1.696353],accel_mss,speed_ms,0,blend_radius_m)
    |   movel([0.127108, -1.307780, -2.618438, -0.786170, 1.570796, 1.697905],accel_mss,speed_ms,0,blend_radius_m)
    |   movel([0.127545, -1.307495, -2.618611, -0.786283, 1.570796, 1.698341],accel_mss,speed_ms,0,blend_radius_m)
    |   movel([0.127946, -1.307258, -2.618755, -0.786376, 1.570796, 1.698743],accel_mss,speed_ms,0,blend_radius_m)
    |   movel([0.128280, -1.307076, -2.618865, -0.786448, 1.570796, 1.699076],accel_mss,speed_ms,0,blend_radius_m)
    |   movel([0.128628, -1.307153, -2.618818, -0.786417, 1.570796, 1.699424],accel_mss,speed_ms,0,blend_radius_m)
    |   movel([0.128839, -1.307535, -2.618587, -0.786267, 1.570796, 1.699635],accel_mss,speed_ms,0,blend_radius_m)
    |   movel([0.129021, -1.308076, -2.618259, -0.786054, 1.570796, 1.699817],accel_mss,speed_ms,0,blend_radius_m)
    |   movel([0.129150, -1.308744, -2.617854, -0.785791, 1.570796, 1.699946],accel_mss,speed_ms,0,blend_radius_m)
    |   movel([0.129190, -1.309116, -2.617628, -0.785645, 1.570796, 1.699986],accel_mss,speed_ms,0,blend_radius_m)
    |   movel([0.129214, -1.309521, -2.617382, -0.785486, 1.570796, 1.700010],accel_mss,speed_ms,0,blend_radius_m)
    |   movel([0.129219, -1.309896, -2.617153, -0.785340, 1.570796, 1.700016],accel_mss,speed_ms,0,blend_radius_m)
    |   movel([0.129197, -1.310174, -2.616984, -0.785231, 1.570796, 1.699993],accel_mss,speed_ms,0,blend_radius_m)
    |   movel([0.129135, -1.310513, -2.616777, -0.785099, 1.570796, 1.699931],accel_mss,speed_ms,0,blend_radius_m)
    |   movel([0.128867, -1.310967, -2.616500, -0.784921, 1.570796, 1.699663],accel_mss,speed_ms,0,blend_radius_m)
    |   movel([0.128512, -1.311321, -2.616284, -0.784783, 1.570796, 1.699309],accel_mss,speed_ms,0,blend_radius_m)
    |   movel([0.127395, -1.312243, -2.615721, -0.784425, 1.570796, 1.698191],accel_mss,speed_ms,0,blend_radius_m)
    |   movel([0.125883, -1.313239, -2.615111, -0.784040, 1.570796, 1.696679],accel_mss,speed_ms,0,blend_radius_m)
    |   movel([0.124104, -1.314236, -2.614498, -0.783654, 1.570796, 1.694900],accel_mss,speed_ms,0,blend_radius_m)
    |   movel([0.122151, -1.315183, -2.613916, -0.783290, 1.570796, 1.692947],accel_mss,speed_ms,0,blend_radius_m)
    |   movel([0.120338, -1.315896, -2.613477, -0.783016, 1.570796, 1.691135],accel_mss,speed_ms,0,blend_radius_m)
    |   movel([0.117897, -1.316665, -2.613002, -0.782722, 1.570796, 1.688693],accel_mss,speed_ms,0,blend_radius_m)
    |   movel([0.115471, -1.317316, -2.612600, -0.782474, 1.570796, 1.686267],accel_mss,speed_ms,0,blend_radius_m)
    |   movel([0.113699, -1.317650, -2.612393, -0.782346, 1.570796, 1.684496],accel_mss,speed_ms,0,blend_radius_m)
    |   movel([0.112470, -1.317775, -2.612315, -0.782298, 1.570796, 1.683266],accel_mss,speed_ms,0,blend_radius_m)
    |   movel([0.111390, -1.317822, -2.612286, -0.782281, 1.570796, 1.682186],accel_mss,speed_ms,0,blend_radius_m)
    |   movel([0.110434, -1.317784, -2.612310, -0.782295, 1.570796, 1.681231],accel_mss,speed_ms,0,blend_radius_m)
    |   movel([0.109566, -1.317665, -2.612384, -0.782341, 1.570796, 1.680362],accel_mss,speed_ms,0,blend_radius_m)
    |   movel([0.108954, -1.317503, -2.612484, -0.782402, 1.570796, 1.679750],accel_mss,speed_ms,0,blend_radius_m)
    |   movel([0.108633, -1.317305, -2.612607, -0.782478, 1.570796, 1.679430],accel_mss,speed_ms,0,blend_radius_m)
    |   movel([0.108500, -1.317001, -2.612794, -0.782594, 1.570796, 1.679296],accel_mss,speed_ms,0,blend_radius_m)
    |   movel([0.108505, -1.316513, -2.613096, -0.782780, 1.570796, 1.679302],accel_mss,speed_ms,0,blend_radius_m)
    |   movel([0.108642, -1.315869, -2.613493, -0.783027, 1.570796, 1.679438],accel_mss,speed_ms,0,blend_radius_m)
    |   movel([0.108950, -1.314910, -2.614084, -0.783395, 1.570796, 1.679746],accel_mss,speed_ms,0,blend_radius_m)
    |   movel([0.109310, -1.313954, -2.614672, -0.783763, 1.570796, 1.680106],accel_mss,speed_ms,0,blend_radius_m)
    |   movel([0.109607, -1.313358, -2.615038, -0.783994, 1.570796, 1.680404],accel_mss,speed_ms,0,blend_radius_m)
    |   movel([0.109887, -1.312990, -2.615263, -0.784136, 1.570796, 1.680684],accel_mss,speed_ms,0,blend_radius_m)
    |   movel([0.110189, -1.312787, -2.615388, -0.784214, 1.570796, 1.680985],accel_mss,speed_ms,0,blend_radius_m)
    |   movel([0.110573, -1.312713, -2.615433, -0.784243, 1.570796, 1.681369],accel_mss,speed_ms,0,blend_radius_m)
    |   movel([0.111158, -1.312760, -2.615404, -0.784225, 1.570796, 1.681955],accel_mss,speed_ms,0,blend_radius_m)
    |   movel([0.112640, -1.312796, -2.615382, -0.784211, 1.570796, 1.683436],accel_mss,speed_ms,0,blend_radius_m)
    |   movel([0.114628, -1.312529, -2.615545, -0.784314, 1.570796, 1.685424],accel_mss,speed_ms,0,blend_radius_m)
    |   movel([0.116962, -1.312002, -2.615868, -0.784519, 1.570796, 1.687758],accel_mss,speed_ms,0,blend_radius_m)
    |   movel([0.119512, -1.311234, -2.616337, -0.784817, 1.570796, 1.690308],accel_mss,speed_ms,0,blend_radius_m)
    |   movel([0.121968, -1.310364, -2.616868, -0.785157, 1.570796, 1.692765],accel_mss,speed_ms,0,blend_radius_m)
    |   speed_ms = 0.003
    |   movel([0.121968, -1.313835, -2.618471, -0.780083, 1.570796, 1.692765],accel_mss,speed_ms,0,blend_radius_m)
    |   speed_ms = 0.007
    |   movel([0.123908, -1.313035, -2.618961, -0.780394, 1.570796, 1.694704],accel_mss,speed_ms,0,blend_radius_m)
    |   movel([0.125557, -1.312206, -2.619467, -0.780716, 1.570796, 1.696353],accel_mss,speed_ms,0,blend_radius_m)
    |   movel([0.127108, -1.311257, -2.620046, -0.781087, 1.570796, 1.697905],accel_mss,speed_ms,0,blend_radius_m)
    |   movel([0.127545, -1.310973, -2.620219, -0.781198, 1.570796, 1.698341],accel_mss,speed_ms,0,blend_radius_m)
    |   movel([0.127946, -1.310736, -2.620363, -0.781290, 1.570796, 1.698743],accel_mss,speed_ms,0,blend_radius_m)
    |   movel([0.128280, -1.310554, -2.620473, -0.781361, 1.570796, 1.699076],accel_mss,speed_ms,0,blend_radius_m)
    |   movel([0.128628, -1.310631, -2.620426, -0.781331, 1.570796, 1.699424],accel_mss,speed_ms,0,blend_radius_m)
    |   movel([0.128839, -1.311012, -2.620195, -0.781182, 1.570796, 1.699635],accel_mss,speed_ms,0,blend_radius_m)
    |   movel([0.129021, -1.311552, -2.619866, -0.780971, 1.570796, 1.699817],accel_mss,speed_ms,0,blend_radius_m)
    |   movel([0.129150, -1.312218, -2.619459, -0.780711, 1.570796, 1.699946],accel_mss,speed_ms,0,blend_radius_m)
    |   movel([0.129190, -1.312590, -2.619232, -0.780567, 1.570796, 1.699986],accel_mss,speed_ms,0,blend_radius_m)
    |   movel([0.129214, -1.312993, -2.618986, -0.780410, 1.570796, 1.700010],accel_mss,speed_ms,0,blend_radius_m)
    |   movel([0.129219, -1.313368, -2.618757, -0.780264, 1.570796, 1.700016],accel_mss,speed_ms,0,blend_radius_m)
    |   movel([0.129197, -1.313645, -2.618587, -0.780157, 1.570796, 1.699993],accel_mss,speed_ms,0,blend_radius_m)
    |   movel([0.129135, -1.313983, -2.618380, -0.780026, 1.570796, 1.699931],accel_mss,speed_ms,0,blend_radius_m)
    |   movel([0.128867, -1.314437, -2.618102, -0.779850, 1.570796, 1.699663],accel_mss,speed_ms,0,blend_radius_m)
    |   movel([0.128512, -1.314790, -2.617885, -0.779714, 1.570796, 1.699309],accel_mss,speed_ms,0,blend_radius_m)
    |   movel([0.127395, -1.315709, -2.617320, -0.779359, 1.570796, 1.698191],accel_mss,speed_ms,0,blend_radius_m)
    |   movel([0.125883, -1.316702, -2.616709, -0.778978, 1.570796, 1.696679],accel_mss,speed_ms,0,blend_radius_m)
    |   movel([0.124104, -1.317698, -2.616095, -0.778597, 1.570796, 1.694900],accel_mss,speed_ms,0,blend_radius_m)
    |   movel([0.122151, -1.318642, -2.615511, -0.778236, 1.570796, 1.692947],accel_mss,speed_ms,0,blend_radius_m)
    |   movel([0.120338, -1.319353, -2.615070, -0.777965, 1.570796, 1.691135],accel_mss,speed_ms,0,blend_radius_m)
    |   movel([0.117897, -1.320120, -2.614594, -0.777674, 1.570796, 1.688693],accel_mss,speed_ms,0,blend_radius_m)
    |   movel([0.115471, -1.320770, -2.614191, -0.777428, 1.570796, 1.686267],accel_mss,speed_ms,0,blend_radius_m)
    |   movel([0.113699, -1.321104, -2.613983, -0.777302, 1.570796, 1.684496],accel_mss,speed_ms,0,blend_radius_m)
    |   movel([0.112470, -1.321228, -2.613906, -0.777255, 1.570796, 1.683266],accel_mss,speed_ms,0,blend_radius_m)
    |   movel([0.111390, -1.321275, -2.613877, -0.777238, 1.570796, 1.682186],accel_mss,speed_ms,0,blend_radius_m)
    |   movel([0.110434, -1.321237, -2.613900, -0.777252, 1.570796, 1.681231],accel_mss,speed_ms,0,blend_radius_m)
    |   movel([0.109566, -1.321118, -2.613974, -0.777297, 1.570796, 1.680362],accel_mss,speed_ms,0,blend_radius_m)
    |   movel([0.108954, -1.320956, -2.614075, -0.777358, 1.570796, 1.679750],accel_mss,speed_ms,0,blend_radius_m)
    |   movel([0.108633, -1.320759, -2.614198, -0.777433, 1.570796, 1.679430],accel_mss,speed_ms,0,blend_radius_m)
    |   movel([0.108500, -1.320456, -2.614386, -0.777547, 1.570796, 1.679296],accel_mss,speed_ms,0,blend_radius_m)
    |   movel([0.108505, -1.319969, -2.614688, -0.777732, 1.570796, 1.679302],accel_mss,speed_ms,0,blend_radius_m)
    |   movel([0.108642, -1.319327, -2.615087, -0.777976, 1.570796, 1.679438],accel_mss,speed_ms,0,blend_radius_m)
    |   movel([0.108950, -1.318370, -2.615679, -0.778340, 1.570796, 1.679746],accel_mss,speed_ms,0,blend_radius_m)
    |   movel([0.109310, -1.317416, -2.616269, -0.778704, 1.570796, 1.680106],accel_mss,speed_ms,0,blend_radius_m)
    |   movel([0.109607, -1.316821, -2.616636, -0.778932, 1.570796, 1.680404],accel_mss,speed_ms,0,blend_radius_m)
    |   movel([0.109887, -1.316454, -2.616862, -0.779073, 1.570796, 1.680684],accel_mss,speed_ms,0,blend_radius_m)
    |   movel([0.110189, -1.316252, -2.616986, -0.779151, 1.570796, 1.680985],accel_mss,speed_ms,0,blend_radius_m)
    |   movel([0.110573, -1.316178, -2.617032, -0.779179, 1.570796, 1.681369],accel_mss,speed_ms,0,blend_radius_m)
    |   movel([0.111158, -1.316225, -2.617003, -0.779161, 1.570796, 1.681955],accel_mss,speed_ms,0,blend_radius_m)
    |   movel([0.112640, -1.316260, -2.616981, -0.779147, 1.570796, 1.683436],accel_mss,speed_ms,0,blend_radius_m)
    |   movel([0.114628, -1.315995, -2.617145, -0.779250, 1.570796, 1.685424],accel_mss,speed_ms,0,blend_radius_m)
    |   movel([0.116962, -1.315469, -2.617468, -0.779452, 1.570796, 1.687758],accel_mss,speed_ms,0,blend_radius_m)
    |   movel([0.119512, -1.314703, -2.617939, -0.779748, 1.570796, 1.690308],accel_mss,speed_ms,0,blend_radius_m)
    |   movel([0.121968, -1.313835, -2.618471, -0.780083, 1.570796, 1.692765],accel_mss,speed_ms,0,blend_radius_m)
    |   speed_ms = 0.003
    |   movel([0.121968, -1.300115, -2.612010, -0.800264, 1.570796, 1.692765],accel_mss,speed_ms,0,blend_radius_m)
    |   speed_ms = 1.000
    |   movel([0.121968, -1.273957, -2.598699, -0.839733, 1.570796, 1.692765],accel_mss,speed_ms,0,blend_radius_m)
    |   movel([0.131398, -1.269919, -2.601026, -0.841444, 1.570796, 1.702195],accel_mss,speed_ms,0,blend_radius_m)
    |   movel([0.131398, -1.296135, -2.614389, -0.801865, 1.570796, 1.702195],accel_mss,speed_ms,0,blend_radius_m)
    |   speed_ms = 0.003
    |   movel([0.131398, -1.306410, -2.619268, -0.786711, 1.570796, 1.702195],accel_mss,speed_ms,0,blend_radius_m)
    |   speed_ms = 0.007
    |   movel([0.131479, -1.305951, -2.619545, -0.786893, 1.570796, 1.702275],accel_mss,speed_ms,0,blend_radius_m)
    |   movel([0.131727, -1.305647, -2.619728, -0.787013, 1.570796, 1.702523],accel_mss,speed_ms,0,blend_radius_m)
    |   movel([0.132252, -1.305356, -2.619904, -0.787129, 1.570796, 1.703049],accel_mss,speed_ms,0,blend_radius_m)
    |   movel([0.132772, -1.305193, -2.620002, -0.787194, 1.570796, 1.703568],accel_mss,speed_ms,0,blend_radius_m)
    |   movel([0.133097, -1.305234, -2.619977, -0.787178, 1.570796, 1.703893],accel_mss,speed_ms,0,blend_radius_m)
    |   movel([0.133324, -1.305510, -2.619811, -0.787068, 1.570796, 1.704120],accel_mss,speed_ms,0,blend_radius_m)
    |   movel([0.133550, -1.306174, -2.619410, -0.786805, 1.570796, 1.704347],accel_mss,speed_ms,0,blend_radius_m)
    |   movel([0.133749, -1.306964, -2.618933, -0.786492, 1.570796, 1.704546],accel_mss,speed_ms,0,blend_radius_m)
    |   movel([0.133844, -1.307602, -2.618546, -0.786240, 1.570796, 1.704640],accel_mss,speed_ms,0,blend_radius_m)
    |   movel([0.133851, -1.308225, -2.618169, -0.785995, 1.570796, 1.704648],accel_mss,speed_ms,0,blend_radius_m)
    |   movel([0.133785, -1.308965, -2.617720, -0.785705, 1.570796, 1.704581],accel_mss,speed_ms,0,blend_radius_m)
    |   movel([0.133710, -1.309445, -2.617428, -0.785516, 1.570796, 1.704506],accel_mss,speed_ms,0,blend_radius_m)
    |   movel([0.133518, -1.309877, -2.617165, -0.785347, 1.570796, 1.704315],accel_mss,speed_ms,0,blend_radius_m)
    |   movel([0.132924, -1.310334, -2.616886, -0.785168, 1.570796, 1.703720],accel_mss,speed_ms,0,blend_radius_m)
    |   movel([0.132460, -1.310561, -2.616748, -0.785080, 1.570796, 1.703256],accel_mss,speed_ms,0,blend_radius_m)
    |   movel([0.132040, -1.310699, -2.616664, -0.785026, 1.570796, 1.702837],accel_mss,speed_ms,0,blend_radius_m)
    |   movel([0.131735, -1.310606, -2.616721, -0.785062, 1.570796, 1.702532],accel_mss,speed_ms,0,blend_radius_m)
    |   movel([0.131676, -1.310395, -2.616849, -0.785145, 1.570796, 1.702472],accel_mss,speed_ms,0,blend_radius_m)
    |   movel([0.131627, -1.310128, -2.617012, -0.785249, 1.570796, 1.702423],accel_mss,speed_ms,0,blend_radius_m)
    |   movel([0.131602, -1.309826, -2.617196, -0.785367, 1.570796, 1.702398],accel_mss,speed_ms,0,blend_radius_m)
    |   movel([0.131582, -1.309429, -2.617437, -0.785522, 1.570796, 1.702379],accel_mss,speed_ms,0,blend_radius_m)
    |   movel([0.131548, -1.308837, -2.617798, -0.785755, 1.570796, 1.702344],accel_mss,speed_ms,0,blend_radius_m)
    |   movel([0.131505, -1.308178, -2.618197, -0.786014, 1.570796, 1.702301],accel_mss,speed_ms,0,blend_radius_m)
    |   movel([0.131461, -1.307540, -2.618584, -0.786265, 1.570796, 1.702257],accel_mss,speed_ms,0,blend_radius_m)
    |   movel([0.131398, -1.306410, -2.619268, -0.786711, 1.570796, 1.702195],accel_mss,speed_ms,0,blend_radius_m)
    |   speed_ms = 0.003
    |   movel([0.131398, -1.309889, -2.620877, -0.781622, 1.570796, 1.702195],accel_mss,speed_ms,0,blend_radius_m)
    |   speed_ms = 0.007
    |   movel([0.131479, -1.309432, -2.621155, -0.781802, 1.570796, 1.702275],accel_mss,speed_ms,0,blend_radius_m)
    |   movel([0.131727, -1.309129, -2.621339, -0.781921, 1.570796, 1.702523],accel_mss,speed_ms,0,blend_radius_m)
    |   movel([0.132252, -1.308838, -2.621515, -0.782036, 1.570796, 1.703049],accel_mss,speed_ms,0,blend_radius_m)
    |   movel([0.132772, -1.308675, -2.621614, -0.782100, 1.570796, 1.703568],accel_mss,speed_ms,0,blend_radius_m)
    |   movel([0.133097, -1.308716, -2.621589, -0.782084, 1.570796, 1.703893],accel_mss,speed_ms,0,blend_radius_m)
    |   movel([0.133324, -1.308991, -2.621422, -0.781975, 1.570796, 1.704120],accel_mss,speed_ms,0,blend_radius_m)
    |   movel([0.133550, -1.309654, -2.621020, -0.781715, 1.570796, 1.704347],accel_mss,speed_ms,0,blend_radius_m)
    |   movel([0.133749, -1.310443, -2.620541, -0.781405, 1.570796, 1.704546],accel_mss,speed_ms,0,blend_radius_m)
    |   movel([0.133844, -1.311079, -2.620154, -0.781156, 1.570796, 1.704640],accel_mss,speed_ms,0,blend_radius_m)
    |   movel([0.133851, -1.311701, -2.619775, -0.780913, 1.570796, 1.704648],accel_mss,speed_ms,0,blend_radius_m)
    |   movel([0.133785, -1.312438, -2.619325, -0.780626, 1.570796, 1.704581],accel_mss,speed_ms,0,blend_radius_m)
    |   movel([0.133710, -1.312917, -2.619032, -0.780439, 1.570796, 1.704506],accel_mss,speed_ms,0,blend_radius_m)
    |   movel([0.133518, -1.313349, -2.618769, -0.780272, 1.570796, 1.704315],accel_mss,speed_ms,0,blend_radius_m)
    |   movel([0.132924, -1.313805, -2.618489, -0.780095, 1.570796, 1.703720],accel_mss,speed_ms,0,blend_radius_m)
    |   movel([0.132460, -1.314031, -2.618350, -0.780007, 1.570796, 1.703256],accel_mss,speed_ms,0,blend_radius_m)
    |   movel([0.132040, -1.314168, -2.618266, -0.779954, 1.570796, 1.702837],accel_mss,speed_ms,0,blend_radius_m)
    |   movel([0.131735, -1.314076, -2.618323, -0.779990, 1.570796, 1.702532],accel_mss,speed_ms,0,blend_radius_m)
    |   movel([0.131676, -1.313866, -2.618452, -0.780071, 1.570796, 1.702472],accel_mss,speed_ms,0,blend_radius_m)
    |   movel([0.131627, -1.313599, -2.618615, -0.780175, 1.570796, 1.702423],accel_mss,speed_ms,0,blend_radius_m)
    |   movel([0.131602, -1.313298, -2.618799, -0.780292, 1.570796, 1.702398],accel_mss,speed_ms,0,blend_radius_m)
    |   movel([0.131582, -1.312902, -2.619042, -0.780445, 1.570796, 1.702379],accel_mss,speed_ms,0,blend_radius_m)
    |   movel([0.131548, -1.312311, -2.619403, -0.780675, 1.570796, 1.702344],accel_mss,speed_ms,0,blend_radius_m)
    |   movel([0.131505, -1.311654, -2.619804, -0.780932, 1.570796, 1.702301],accel_mss,speed_ms,0,blend_radius_m)
    |   movel([0.131461, -1.311017, -2.620191, -0.781180, 1.570796, 1.702257],accel_mss,speed_ms,0,blend_radius_m)
    |   movel([0.131398, -1.309889, -2.620877, -0.781622, 1.570796, 1.702195],accel_mss,speed_ms,0,blend_radius_m)
    |   speed_ms = 0.003
    |   movel([0.131398, -1.296135, -2.614389, -0.801865, 1.570796, 1.702195],accel_mss,speed_ms,0,blend_radius_m)
    |   speed_ms = 1.000
    |   movel([0.131398, -1.269919, -2.601026, -0.841444, 1.570796, 1.702195],accel_mss,speed_ms,0,blend_radius_m)
    |   movel([0.130856, -1.269619, -2.601198, -0.841572, 1.570796, 1.701652],accel_mss,speed_ms,0,blend_radius_m)
    |   movel([0.130856, -1.295838, -2.614566, -0.801985, 1.570796, 1.701652],accel_mss,speed_ms,0,blend_radius_m)
    |   speed_ms = 0.003
    |   movel([0.130856, -1.306115, -2.619446, -0.786828, 1.570796, 1.701652],accel_mss,speed_ms,0,blend_radius_m)
    |   speed_ms = 0.007
    |   movel([0.131011, -1.307925, -2.618350, -0.786113, 1.570796, 1.701808],accel_mss,speed_ms,0,blend_radius_m)
    |   movel([0.131148, -1.310741, -2.616638, -0.785010, 1.570796, 1.701944],accel_mss,speed_ms,0,blend_radius_m)
    |   movel([0.131240, -1.313539, -2.614926, -0.783923, 1.570796, 1.702036],accel_mss,speed_ms,0,blend_radius_m)
    |   movel([0.131227, -1.315239, -2.613882, -0.783269, 1.570796, 1.702023],accel_mss,speed_ms,0,blend_radius_m)
    |   movel([0.131217, -1.315548, -2.613691, -0.783150, 1.570796, 1.702014],accel_mss,speed_ms,0,blend_radius_m)
    |   movel([0.131173, -1.315815, -2.613527, -0.783048, 1.570796, 1.701969],accel_mss,speed_ms,0,blend_radius_m)
    |   movel([0.130301, -1.316397, -2.613168, -0.782825, 1.570796, 1.701098],accel_mss,speed_ms,0,blend_radius_m)
    |   movel([0.125673, -1.317927, -2.612221, -0.782241, 1.570796, 1.696469],accel_mss,speed_ms,0,blend_radius_m)
    |   movel([0.120471, -1.319590, -2.611190, -0.781610, 1.570796, 1.691267],accel_mss,speed_ms,0,blend_radius_m)
    |   movel([0.114839, -1.321304, -2.610122, -0.780963, 1.570796, 1.685636],accel_mss,speed_ms,0,blend_radius_m)
    |   movel([0.110155, -1.322696, -2.609252, -0.780441, 1.570796, 1.680951],accel_mss,speed_ms,0,blend_radius_m)
    |   movel([0.107702, -1.323389, -2.608818, -0.780182, 1.570796, 1.678499],accel_mss,speed_ms,0,blend_radius_m)
    |   movel([0.106178, -1.323770, -2.608580, -0.780040, 1.570796, 1.676974],accel_mss,speed_ms,0,blend_radius_m)
    |   movel([0.105794, -1.323707, -2.608619, -0.780063, 1.570796, 1.676590],accel_mss,speed_ms,0,blend_radius_m)
    |   movel([0.105803, -1.322985, -2.609071, -0.780333, 1.570796, 1.676600],accel_mss,speed_ms,0,blend_radius_m)
    |   movel([0.105951, -1.322098, -2.609626, -0.780665, 1.570796, 1.676748],accel_mss,speed_ms,0,blend_radius_m)
    |   movel([0.106248, -1.320539, -2.610599, -0.781251, 1.570796, 1.677044],accel_mss,speed_ms,0,blend_radius_m)
    |   movel([0.107313, -1.315582, -2.613670, -0.783137, 1.570796, 1.678109],accel_mss,speed_ms,0,blend_radius_m)
    |   movel([0.108622, -1.310362, -2.616870, -0.785158, 1.570796, 1.679418],accel_mss,speed_ms,0,blend_radius_m)
    |   movel([0.109963, -1.305509, -2.619812, -0.787068, 1.570796, 1.680759],accel_mss,speed_ms,0,blend_radius_m)
    |   movel([0.110603, -1.304268, -2.620559, -0.787562, 1.570796, 1.681400],accel_mss,speed_ms,0,blend_radius_m)
    |   movel([0.111988, -1.303208, -2.621196, -0.787985, 1.570796, 1.682784],accel_mss,speed_ms,0,blend_radius_m)
    |   movel([0.117483, -1.301191, -2.622403, -0.788794, 1.570796, 1.688279],accel_mss,speed_ms,0,blend_radius_m)
    |   movel([0.123023, -1.299415, -2.623463, -0.789511, 1.570796, 1.693820],accel_mss,speed_ms,0,blend_radius_m)
    |   movel([0.127025, -1.298536, -2.623985, -0.789867, 1.570796, 1.697822],accel_mss,speed_ms,0,blend_radius_m)
    |   movel([0.128125, -1.298410, -2.624060, -0.789919, 1.570796, 1.698921],accel_mss,speed_ms,0,blend_radius_m)
    |   movel([0.128706, -1.298444, -2.624040, -0.789905, 1.570796, 1.699503],accel_mss,speed_ms,0,blend_radius_m)
    |   movel([0.129058, -1.298646, -2.623920, -0.789823, 1.570796, 1.699855],accel_mss,speed_ms,0,blend_radius_m)
    |   movel([0.129325, -1.299072, -2.623667, -0.789650, 1.570796, 1.700122],accel_mss,speed_ms,0,blend_radius_m)
    |   movel([0.129761, -1.300339, -2.622912, -0.789138, 1.570796, 1.700558],accel_mss,speed_ms,0,blend_radius_m)
    |   movel([0.130190, -1.302093, -2.621864, -0.788432, 1.570796, 1.700986],accel_mss,speed_ms,0,blend_radius_m)
    |   movel([0.130571, -1.304084, -2.620670, -0.787635, 1.570796, 1.701368],accel_mss,speed_ms,0,blend_radius_m)
    |   movel([0.130856, -1.306115, -2.619446, -0.786828, 1.570796, 1.701652],accel_mss,speed_ms,0,blend_radius_m)
    |   speed_ms = 0.003
    |   movel([0.130856, -1.309595, -2.621056, -0.781738, 1.570796, 1.701652],accel_mss,speed_ms,0,blend_radius_m)
    |   speed_ms = 0.007
    |   movel([0.131011, -1.311402, -2.619957, -0.781030, 1.570796, 1.701808],accel_mss,speed_ms,0,blend_radius_m)
    |   movel([0.131148, -1.314211, -2.618241, -0.779938, 1.570796, 1.701944],accel_mss,speed_ms,0,blend_radius_m)
    |   movel([0.131240, -1.317002, -2.616524, -0.778863, 1.570796, 1.702036],accel_mss,speed_ms,0,blend_radius_m)
    |   movel([0.131227, -1.318698, -2.615476, -0.778215, 1.570796, 1.702023],accel_mss,speed_ms,0,blend_radius_m)
    |   movel([0.131217, -1.319007, -2.615285, -0.778097, 1.570796, 1.702014],accel_mss,speed_ms,0,blend_radius_m)
    |   movel([0.131173, -1.319272, -2.615120, -0.777996, 1.570796, 1.701969],accel_mss,speed_ms,0,blend_radius_m)
    |   movel([0.130301, -1.319853, -2.614760, -0.777776, 1.570796, 1.701098],accel_mss,speed_ms,0,blend_radius_m)
    |   movel([0.125673, -1.321380, -2.613811, -0.777198, 1.570796, 1.696469],accel_mss,speed_ms,0,blend_radius_m)
    |   movel([0.120471, -1.323038, -2.612777, -0.776574, 1.570796, 1.691267],accel_mss,speed_ms,0,blend_radius_m)
    |   movel([0.114839, -1.324749, -2.611706, -0.775934, 1.570796, 1.685636],accel_mss,speed_ms,0,blend_radius_m)
    |   movel([0.110155, -1.326137, -2.610834, -0.775418, 1.570796, 1.680951],accel_mss,speed_ms,0,blend_radius_m)
    |   movel([0.107702, -1.326828, -2.610399, -0.775162, 1.570796, 1.678499],accel_mss,speed_ms,0,blend_radius_m)
    |   movel([0.106178, -1.327208, -2.610160, -0.775021, 1.570796, 1.676974],accel_mss,speed_ms,0,blend_radius_m)
    |   movel([0.105794, -1.327146, -2.610199, -0.775044, 1.570796, 1.676590],accel_mss,speed_ms,0,blend_radius_m)
    |   movel([0.105803, -1.326426, -2.610652, -0.775311, 1.570796, 1.676600],accel_mss,speed_ms,0,blend_radius_m)
    |   movel([0.105951, -1.325541, -2.611209, -0.775639, 1.570796, 1.676748],accel_mss,speed_ms,0,blend_radius_m)
    |   movel([0.106248, -1.323986, -2.612184, -0.776219, 1.570796, 1.677044],accel_mss,speed_ms,0,blend_radius_m)
    |   movel([0.107313, -1.319041, -2.615264, -0.778084, 1.570796, 1.678109],accel_mss,speed_ms,0,blend_radius_m)
    |   movel([0.108622, -1.313832, -2.618473, -0.780084, 1.570796, 1.679418],accel_mss,speed_ms,0,blend_radius_m)
    |   movel([0.109963, -1.308991, -2.621423, -0.781976, 1.570796, 1.680759],accel_mss,speed_ms,0,blend_radius_m)
    |   movel([0.110603, -1.307752, -2.622172, -0.782464, 1.570796, 1.681400],accel_mss,speed_ms,0,blend_radius_m)
    |   movel([0.111988, -1.306695, -2.622811, -0.782883, 1.570796, 1.682784],accel_mss,speed_ms,0,blend_radius_m)
    |   movel([0.117483, -1.304683, -2.624022, -0.783684, 1.570796, 1.688279],accel_mss,speed_ms,0,blend_radius_m)
    |   movel([0.123023, -1.302911, -2.625084, -0.784394, 1.570796, 1.693820],accel_mss,speed_ms,0,blend_radius_m)
    |   movel([0.127025, -1.302034, -2.625608, -0.784747, 1.570796, 1.697822],accel_mss,speed_ms,0,blend_radius_m)
    |   movel([0.128125, -1.301908, -2.625683, -0.784798, 1.570796, 1.698921],accel_mss,speed_ms,0,blend_radius_m)
    |   movel([0.128706, -1.301942, -2.625663, -0.784784, 1.570796, 1.699503],accel_mss,speed_ms,0,blend_radius_m)
    |   movel([0.129058, -1.302144, -2.625543, -0.784703, 1.570796, 1.699855],accel_mss,speed_ms,0,blend_radius_m)
    |   movel([0.129325, -1.302568, -2.625289, -0.784532, 1.570796, 1.700122],accel_mss,speed_ms,0,blend_radius_m)
    |   movel([0.129761, -1.303833, -2.624532, -0.784024, 1.570796, 1.700558],accel_mss,speed_ms,0,blend_radius_m)
    |   movel([0.130190, -1.305582, -2.623481, -0.783325, 1.570796, 1.700986],accel_mss,speed_ms,0,blend_radius_m)
    |   movel([0.130571, -1.307569, -2.622283, -0.782537, 1.570796, 1.701368],accel_mss,speed_ms,0,blend_radius_m)
    |   movel([0.130856, -1.309595, -2.621056, -0.781738, 1.570796, 1.701652],accel_mss,speed_ms,0,blend_radius_m)
    |   speed_ms = 0.003
    |   movel([0.130856, -1.295838, -2.614566, -0.801985, 1.570796, 1.701652],accel_mss,speed_ms,0,blend_radius_m)
    |   speed_ms = 1.000
    |   movel([0.130856, -1.269619, -2.601198, -0.841572, 1.570796, 1.701652],accel_mss,speed_ms,0,blend_radius_m)
    |   movel([0.130531, -1.280367, -2.594964, -0.837058, 1.570796, 1.701327],accel_mss,speed_ms,0,blend_radius_m)
    |   movel([0.130531, -1.306432, -2.608191, -0.797766, 1.570796, 1.701327],accel_mss,speed_ms,0,blend_radius_m)
    |   speed_ms = 0.003
    |   movel([0.130531, -1.316639, -2.613018, -0.782732, 1.570796, 1.701327],accel_mss,speed_ms,0,blend_radius_m)
    |   speed_ms = 0.007
    |   movel([0.131235, -1.316442, -2.613140, -0.782807, 1.570796, 1.702031],accel_mss,speed_ms,0,blend_radius_m)
    |   movel([0.131541, -1.316548, -2.613074, -0.782767, 1.570796, 1.702337],accel_mss,speed_ms,0,blend_radius_m)
    |   movel([0.131627, -1.316974, -2.612811, -0.782604, 1.570796, 1.702424],accel_mss,speed_ms,0,blend_radius_m)
    |   movel([0.131494, -1.318238, -2.612029, -0.782122, 1.570796, 1.702291],accel_mss,speed_ms,0,blend_radius_m)
    |   movel([0.131414, -1.318780, -2.611693, -0.781917, 1.570796, 1.702210],accel_mss,speed_ms,0,blend_radius_m)
    |   movel([0.131342, -1.319073, -2.611510, -0.781805, 1.570796, 1.702139],accel_mss,speed_ms,0,blend_radius_m)
    |   movel([0.131110, -1.319399, -2.611308, -0.781682, 1.570796, 1.701906],accel_mss,speed_ms,0,blend_radius_m)
    |   movel([0.130624, -1.319661, -2.611145, -0.781583, 1.570796, 1.701421],accel_mss,speed_ms,0,blend_radius_m)
    |   movel([0.127936, -1.320652, -2.610528, -0.781208, 1.570796, 1.698733],accel_mss,speed_ms,0,blend_radius_m)
    |   movel([0.125277, -1.321610, -2.609931, -0.780848, 1.570796, 1.696074],accel_mss,speed_ms,0,blend_radius_m)
    |   movel([0.123158, -1.322327, -2.609483, -0.780579, 1.570796, 1.693954],accel_mss,speed_ms,0,blend_radius_m)
    |   movel([0.122291, -1.322606, -2.609308, -0.780475, 1.570796, 1.693087],accel_mss,speed_ms,0,blend_radius_m)
    |   movel([0.121350, -1.322916, -2.609114, -0.780359, 1.570796, 1.692146],accel_mss,speed_ms,0,blend_radius_m)
    |   movel([0.120477, -1.323205, -2.608933, -0.780251, 1.570796, 1.691273],accel_mss,speed_ms,0,blend_radius_m)
    |   movel([0.119834, -1.323423, -2.608797, -0.780169, 1.570796, 1.690631],accel_mss,speed_ms,0,blend_radius_m)
    |   movel([0.119284, -1.323604, -2.608683, -0.780102, 1.570796, 1.690080],accel_mss,speed_ms,0,blend_radius_m)
    |   movel([0.118876, -1.323722, -2.608610, -0.780058, 1.570796, 1.689672],accel_mss,speed_ms,0,blend_radius_m)
    |   movel([0.118580, -1.323788, -2.608568, -0.780033, 1.570796, 1.689376],accel_mss,speed_ms,0,blend_radius_m)
    |   movel([0.118701, -1.323511, -2.608742, -0.780136, 1.570796, 1.689498],accel_mss,speed_ms,0,blend_radius_m)
    |   movel([0.119077, -1.323087, -2.609008, -0.780295, 1.570796, 1.689873],accel_mss,speed_ms,0,blend_radius_m)
    |   movel([0.119370, -1.322757, -2.609214, -0.780418, 1.570796, 1.690167],accel_mss,speed_ms,0,blend_radius_m)
    |   movel([0.119620, -1.322278, -2.609514, -0.780598, 1.570796, 1.690416],accel_mss,speed_ms,0,blend_radius_m)
    |   movel([0.119685, -1.321910, -2.609744, -0.780736, 1.570796, 1.690481],accel_mss,speed_ms,0,blend_radius_m)
    |   movel([0.119717, -1.321544, -2.609972, -0.780873, 1.570796, 1.690513],accel_mss,speed_ms,0,blend_radius_m)
    |   movel([0.119567, -1.321184, -2.610197, -0.781008, 1.570796, 1.690364],accel_mss,speed_ms,0,blend_radius_m)
    |   movel([0.119305, -1.320996, -2.610314, -0.781079, 1.570796, 1.690101],accel_mss,speed_ms,0,blend_radius_m)
    |   movel([0.118996, -1.320712, -2.610491, -0.781186, 1.570796, 1.689792],accel_mss,speed_ms,0,blend_radius_m)
    |   movel([0.119567, -1.320254, -2.610776, -0.781359, 1.570796, 1.690363],accel_mss,speed_ms,0,blend_radius_m)
    |   movel([0.121060, -1.319799, -2.611060, -0.781531, 1.570796, 1.691857],accel_mss,speed_ms,0,blend_radius_m)
    |   movel([0.122825, -1.319250, -2.611401, -0.781738, 1.570796, 1.693621],accel_mss,speed_ms,0,blend_radius_m)
    |   movel([0.125783, -1.318274, -2.612006, -0.782109, 1.570796, 1.696580],accel_mss,speed_ms,0,blend_radius_m)
    |   movel([0.128743, -1.317278, -2.612623, -0.782488, 1.570796, 1.699540],accel_mss,speed_ms,0,blend_radius_m)
    |   movel([0.130531, -1.316639, -2.613018, -0.782732, 1.570796, 1.701327],accel_mss,speed_ms,0,blend_radius_m)
    |   speed_ms = 0.003
    |   movel([0.130531, -1.320095, -2.614610, -0.777684, 1.570796, 1.701327],accel_mss,speed_ms,0,blend_radius_m)
    |   speed_ms = 0.007
    |   movel([0.131235, -1.319898, -2.614732, -0.777759, 1.570796, 1.702031],accel_mss,speed_ms,0,blend_radius_m)
    |   movel([0.131541, -1.320004, -2.614667, -0.777719, 1.570796, 1.702337],accel_mss,speed_ms,0,blend_radius_m)
    |   movel([0.131627, -1.320429, -2.614402, -0.777557, 1.570796, 1.702424],accel_mss,speed_ms,0,blend_radius_m)
    |   movel([0.131494, -1.321690, -2.613618, -0.777081, 1.570796, 1.702291],accel_mss,speed_ms,0,blend_radius_m)
    |   movel([0.131414, -1.322230, -2.613281, -0.776877, 1.570796, 1.702210],accel_mss,speed_ms,0,blend_radius_m)
    |   movel([0.131342, -1.322523, -2.613098, -0.776767, 1.570796, 1.702139],accel_mss,speed_ms,0,blend_radius_m)
    |   movel([0.131110, -1.322848, -2.612896, -0.776645, 1.570796, 1.701906],accel_mss,speed_ms,0,blend_radius_m)
    |   movel([0.130624, -1.323110, -2.612732, -0.776547, 1.570796, 1.701421],accel_mss,speed_ms,0,blend_radius_m)
    |   movel([0.127936, -1.324099, -2.612114, -0.776177, 1.570796, 1.698733],accel_mss,speed_ms,0,blend_radius_m)
    |   movel([0.125277, -1.325054, -2.611515, -0.775820, 1.570796, 1.696074],accel_mss,speed_ms,0,blend_radius_m)
    |   movel([0.123158, -1.325769, -2.611066, -0.775554, 1.570796, 1.693954],accel_mss,speed_ms,0,blend_radius_m)
    |   movel([0.122291, -1.326047, -2.610891, -0.775451, 1.570796, 1.693087],accel_mss,speed_ms,0,blend_radius_m)
    |   movel([0.121350, -1.326357, -2.610696, -0.775336, 1.570796, 1.692146],accel_mss,speed_ms,0,blend_radius_m)
    |   movel([0.120477, -1.326645, -2.610514, -0.775229, 1.570796, 1.691273],accel_mss,speed_ms,0,blend_radius_m)
    |   movel([0.119834, -1.326862, -2.610378, -0.775149, 1.570796, 1.690631],accel_mss,speed_ms,0,blend_radius_m)
    |   movel([0.119284, -1.327043, -2.610264, -0.775082, 1.570796, 1.690080],accel_mss,speed_ms,0,blend_radius_m)
    |   movel([0.118876, -1.327160, -2.610190, -0.775039, 1.570796, 1.689672],accel_mss,speed_ms,0,blend_radius_m)
    |   movel([0.118580, -1.327227, -2.610148, -0.775014, 1.570796, 1.689376],accel_mss,speed_ms,0,blend_radius_m)
    |   movel([0.118701, -1.326950, -2.610322, -0.775116, 1.570796, 1.689498],accel_mss,speed_ms,0,blend_radius_m)
    |   movel([0.119077, -1.326527, -2.610589, -0.775273, 1.570796, 1.689873],accel_mss,speed_ms,0,blend_radius_m)
    |   movel([0.119370, -1.326198, -2.610796, -0.775395, 1.570796, 1.690167],accel_mss,speed_ms,0,blend_radius_m)
    |   movel([0.119620, -1.325720, -2.611096, -0.775573, 1.570796, 1.690416],accel_mss,speed_ms,0,blend_radius_m)
    |   movel([0.119685, -1.325353, -2.611327, -0.775709, 1.570796, 1.690481],accel_mss,speed_ms,0,blend_radius_m)
    |   movel([0.119717, -1.324988, -2.611556, -0.775845, 1.570796, 1.690513],accel_mss,speed_ms,0,blend_radius_m)
    |   movel([0.119567, -1.324629, -2.611781, -0.775979, 1.570796, 1.690364],accel_mss,speed_ms,0,blend_radius_m)
    |   movel([0.119305, -1.324442, -2.611899, -0.776049, 1.570796, 1.690101],accel_mss,speed_ms,0,blend_radius_m)
    |   movel([0.118996, -1.324158, -2.612076, -0.776154, 1.570796, 1.689792],accel_mss,speed_ms,0,blend_radius_m)
    |   movel([0.119567, -1.323701, -2.612363, -0.776326, 1.570796, 1.690363],accel_mss,speed_ms,0,blend_radius_m)
    |   movel([0.121060, -1.323247, -2.612646, -0.776496, 1.570796, 1.691857],accel_mss,speed_ms,0,blend_radius_m)
    |   movel([0.122825, -1.322700, -2.612988, -0.776701, 1.570796, 1.693621],accel_mss,speed_ms,0,blend_radius_m)
    |   movel([0.125783, -1.321726, -2.613596, -0.777067, 1.570796, 1.696580],accel_mss,speed_ms,0,blend_radius_m)
    |   movel([0.128743, -1.320732, -2.614214, -0.777443, 1.570796, 1.699540],accel_mss,speed_ms,0,blend_radius_m)
    |   movel([0.130531, -1.320095, -2.614610, -0.777684, 1.570796, 1.701327],accel_mss,speed_ms,0,blend_radius_m)
    |   speed_ms = 0.003
    |   movel([0.130531, -1.306432, -2.608191, -0.797766, 1.570796, 1.701327],accel_mss,speed_ms,0,blend_radius_m)
    |   speed_ms = 1.000
    |   movel([0.130531, -1.280367, -2.594964, -0.837058, 1.570796, 1.701327],accel_mss,speed_ms,0,blend_radius_m)
    |   movel([0.134041, -1.278189, -2.596239, -0.837961, 1.570796, 1.704837],accel_mss,speed_ms,0,blend_radius_m)
    |   movel([0.134041, -1.304285, -2.609494, -0.798609, 1.570796, 1.704837],accel_mss,speed_ms,0,blend_radius_m)
    |   speed_ms = 0.003
    |   movel([0.134041, -1.314507, -2.614332, -0.783550, 1.570796, 1.704837],accel_mss,speed_ms,0,blend_radius_m)
    |   speed_ms = 0.007
    |   movel([0.133922, -1.314134, -2.614561, -0.783694, 1.570796, 1.704718],accel_mss,speed_ms,0,blend_radius_m)
    |   movel([0.133816, -1.313691, -2.614833, -0.783865, 1.570796, 1.704612],accel_mss,speed_ms,0,blend_radius_m)
    |   movel([0.133737, -1.313248, -2.615105, -0.784036, 1.570796, 1.704534],accel_mss,speed_ms,0,blend_radius_m)
    |   movel([0.133705, -1.312880, -2.615331, -0.784178, 1.570796, 1.704501],accel_mss,speed_ms,0,blend_radius_m)
    |   movel([0.133672, -1.312482, -2.615575, -0.784333, 1.570796, 1.704468],accel_mss,speed_ms,0,blend_radius_m)
    |   movel([0.133600, -1.312150, -2.615778, -0.784461, 1.570796, 1.704396],accel_mss,speed_ms,0,blend_radius_m)
    |   movel([0.133482, -1.311864, -2.615953, -0.784573, 1.570796, 1.704279],accel_mss,speed_ms,0,blend_radius_m)
    |   movel([0.133315, -1.311601, -2.616113, -0.784675, 1.570796, 1.704111],accel_mss,speed_ms,0,blend_radius_m)
    |   movel([0.133087, -1.311256, -2.616324, -0.784809, 1.570796, 1.703883],accel_mss,speed_ms,0,blend_radius_m)
    |   movel([0.133002, -1.310974, -2.616496, -0.784919, 1.570796, 1.703798],accel_mss,speed_ms,0,blend_radius_m)
    |   movel([0.133211, -1.310582, -2.616736, -0.785072, 1.570796, 1.704007],accel_mss,speed_ms,0,blend_radius_m)
    |   movel([0.133522, -1.310527, -2.616769, -0.785093, 1.570796, 1.704318],accel_mss,speed_ms,0,blend_radius_m)
    |   movel([0.133930, -1.310895, -2.616544, -0.784950, 1.570796, 1.704727],accel_mss,speed_ms,0,blend_radius_m)
    |   movel([0.134168, -1.311210, -2.616352, -0.784827, 1.570796, 1.704964],accel_mss,speed_ms,0,blend_radius_m)
    |   movel([0.134311, -1.311517, -2.616165, -0.784707, 1.570796, 1.705107],accel_mss,speed_ms,0,blend_radius_m)
    |   movel([0.134387, -1.311901, -2.615930, -0.784558, 1.570796, 1.705183],accel_mss,speed_ms,0,blend_radius_m)
    |   movel([0.134426, -1.312467, -2.615583, -0.784338, 1.570796, 1.705222],accel_mss,speed_ms,0,blend_radius_m)
    |   movel([0.134455, -1.312786, -2.615389, -0.784215, 1.570796, 1.705252],accel_mss,speed_ms,0,blend_radius_m)
    |   movel([0.134534, -1.313187, -2.615143, -0.784060, 1.570796, 1.705331],accel_mss,speed_ms,0,blend_radius_m)
    |   movel([0.134640, -1.313599, -2.614890, -0.783900, 1.570796, 1.705436],accel_mss,speed_ms,0,blend_radius_m)
    |   movel([0.134763, -1.313959, -2.614669, -0.783761, 1.570796, 1.705560],accel_mss,speed_ms,0,blend_radius_m)
    |   movel([0.134892, -1.314355, -2.614426, -0.783609, 1.570796, 1.705688],accel_mss,speed_ms,0,blend_radius_m)
    |   movel([0.135006, -1.314858, -2.614116, -0.783415, 1.570796, 1.705803],accel_mss,speed_ms,0,blend_radius_m)
    |   movel([0.135093, -1.315392, -2.613787, -0.783210, 1.570796, 1.705889],accel_mss,speed_ms,0,blend_radius_m)
    |   movel([0.135137, -1.315883, -2.613485, -0.783021, 1.570796, 1.705933],accel_mss,speed_ms,0,blend_radius_m)
    |   movel([0.135177, -1.316363, -2.613189, -0.782838, 1.570796, 1.705974],accel_mss,speed_ms,0,blend_radius_m)
    |   movel([0.135251, -1.316890, -2.612863, -0.782636, 1.570796, 1.706048],accel_mss,speed_ms,0,blend_radius_m)
    |   movel([0.135343, -1.317384, -2.612557, -0.782448, 1.570796, 1.706140],accel_mss,speed_ms,0,blend_radius_m)
    |   movel([0.135444, -1.317754, -2.612329, -0.782307, 1.570796, 1.706240],accel_mss,speed_ms,0,blend_radius_m)
    |   movel([0.135639, -1.318363, -2.611951, -0.782075, 1.570796, 1.706435],accel_mss,speed_ms,0,blend_radius_m)
    |   movel([0.135633, -1.318671, -2.611760, -0.781958, 1.570796, 1.706429],accel_mss,speed_ms,0,blend_radius_m)
    |   movel([0.135314, -1.318979, -2.611569, -0.781841, 1.570796, 1.706110],accel_mss,speed_ms,0,blend_radius_m)
    |   movel([0.135031, -1.319099, -2.611494, -0.781795, 1.570796, 1.705828],accel_mss,speed_ms,0,blend_radius_m)
    |   movel([0.134712, -1.319109, -2.611488, -0.781792, 1.570796, 1.705508],accel_mss,speed_ms,0,blend_radius_m)
    |   movel([0.134730, -1.318705, -2.611739, -0.781945, 1.570796, 1.705526],accel_mss,speed_ms,0,blend_radius_m)
    |   movel([0.134718, -1.318372, -2.611945, -0.782071, 1.570796, 1.705515],accel_mss,speed_ms,0,blend_radius_m)
    |   movel([0.134682, -1.318089, -2.612121, -0.782179, 1.570796, 1.705478],accel_mss,speed_ms,0,blend_radius_m)
    |   movel([0.134613, -1.317844, -2.612273, -0.782272, 1.570796, 1.705410],accel_mss,speed_ms,0,blend_radius_m)
    |   movel([0.134557, -1.317636, -2.612401, -0.782351, 1.570796, 1.705354],accel_mss,speed_ms,0,blend_radius_m)
    |   movel([0.134502, -1.317270, -2.612628, -0.782491, 1.570796, 1.705299],accel_mss,speed_ms,0,blend_radius_m)
    |   movel([0.134451, -1.316842, -2.612892, -0.782654, 1.570796, 1.705248],accel_mss,speed_ms,0,blend_radius_m)
    |   movel([0.134415, -1.316404, -2.613163, -0.782822, 1.570796, 1.705211],accel_mss,speed_ms,0,blend_radius_m)
    |   movel([0.134367, -1.315933, -2.613454, -0.783002, 1.570796, 1.705164],accel_mss,speed_ms,0,blend_radius_m)
    |   movel([0.134277, -1.315403, -2.613781, -0.783206, 1.570796, 1.705074],accel_mss,speed_ms,0,blend_radius_m)
    |   movel([0.134162, -1.314900, -2.614090, -0.783399, 1.570796, 1.704959],accel_mss,speed_ms,0,blend_radius_m)
    |   movel([0.134041, -1.314507, -2.614332, -0.783550, 1.570796, 1.704837],accel_mss,speed_ms,0,blend_radius_m)
    |   speed_ms = 0.003
    |   movel([0.134041, -1.317968, -2.615928, -0.778493, 1.570796, 1.704837],accel_mss,speed_ms,0,blend_radius_m)
    |   speed_ms = 0.007
    |   movel([0.133922, -1.317596, -2.616157, -0.778635, 1.570796, 1.704718],accel_mss,speed_ms,0,blend_radius_m)
    |   movel([0.133816, -1.317153, -2.616431, -0.778805, 1.570796, 1.704612],accel_mss,speed_ms,0,blend_radius_m)
    |   movel([0.133737, -1.316712, -2.616703, -0.778974, 1.570796, 1.704534],accel_mss,speed_ms,0,blend_radius_m)
    |   movel([0.133705, -1.316344, -2.616929, -0.779115, 1.570796, 1.704501],accel_mss,speed_ms,0,blend_radius_m)
    |   movel([0.133672, -1.315947, -2.617174, -0.779268, 1.570796, 1.704468],accel_mss,speed_ms,0,blend_radius_m)
    |   movel([0.133600, -1.315616, -2.617377, -0.779395, 1.570796, 1.704396],accel_mss,speed_ms,0,blend_radius_m)
    |   movel([0.133482, -1.315331, -2.617553, -0.779505, 1.570796, 1.704279],accel_mss,speed_ms,0,blend_radius_m)
    |   movel([0.133315, -1.315069, -2.617714, -0.779606, 1.570796, 1.704111],accel_mss,speed_ms,0,blend_radius_m)
    |   movel([0.133087, -1.314724, -2.617925, -0.779739, 1.570796, 1.703883],accel_mss,speed_ms,0,blend_radius_m)
    |   movel([0.133002, -1.314443, -2.618098, -0.779848, 1.570796, 1.703798],accel_mss,speed_ms,0,blend_radius_m)
    |   movel([0.133211, -1.314052, -2.618338, -0.779999, 1.570796, 1.704007],accel_mss,speed_ms,0,blend_radius_m)
    |   movel([0.133522, -1.313997, -2.618372, -0.780021, 1.570796, 1.704318],accel_mss,speed_ms,0,blend_radius_m)
    |   movel([0.133930, -1.314364, -2.618146, -0.779878, 1.570796, 1.704727],accel_mss,speed_ms,0,blend_radius_m)
    |   movel([0.134168, -1.314678, -2.617954, -0.779757, 1.570796, 1.704964],accel_mss,speed_ms,0,blend_radius_m)
    |   movel([0.134311, -1.314985, -2.617765, -0.779639, 1.570796, 1.705107],accel_mss,speed_ms,0,blend_radius_m)
    |   movel([0.134387, -1.315368, -2.617530, -0.779491, 1.570796, 1.705183],accel_mss,speed_ms,0,blend_radius_m)
    |   movel([0.134426, -1.315933, -2.617183, -0.779273, 1.570796, 1.705222],accel_mss,speed_ms,0,blend_radius_m)
    |   movel([0.134455, -1.316250, -2.616987, -0.779151, 1.570796, 1.705252],accel_mss,speed_ms,0,blend_radius_m)
    |   movel([0.134534, -1.316651, -2.616741, -0.778998, 1.570796, 1.705331],accel_mss,speed_ms,0,blend_radius_m)
    |   movel([0.134640, -1.317062, -2.616487, -0.778840, 1.570796, 1.705436],accel_mss,speed_ms,0,blend_radius_m)
    |   movel([0.134763, -1.317421, -2.616265, -0.778702, 1.570796, 1.705560],accel_mss,speed_ms,0,blend_radius_m)
    |   movel([0.134892, -1.317816, -2.616022, -0.778551, 1.570796, 1.705688],accel_mss,speed_ms,0,blend_radius_m)
    |   movel([0.135006, -1.318318, -2.615711, -0.778360, 1.570796, 1.705803],accel_mss,speed_ms,0,blend_radius_m)
    |   movel([0.135093, -1.318851, -2.615381, -0.778157, 1.570796, 1.705889],accel_mss,speed_ms,0,blend_radius_m)
    |   movel([0.135137, -1.319340, -2.615078, -0.777970, 1.570796, 1.705933],accel_mss,speed_ms,0,blend_radius_m)
    |   movel([0.135177, -1.319819, -2.614781, -0.777789, 1.570796, 1.705974],accel_mss,speed_ms,0,blend_radius_m)
    |   movel([0.135251, -1.320345, -2.614455, -0.777589, 1.570796, 1.706048],accel_mss,speed_ms,0,blend_radius_m)
    |   movel([0.135343, -1.320838, -2.614148, -0.777403, 1.570796, 1.706140],accel_mss,speed_ms,0,blend_radius_m)
    |   movel([0.135444, -1.321207, -2.613919, -0.777263, 1.570796, 1.706240],accel_mss,speed_ms,0,blend_radius_m)
    |   movel([0.135639, -1.321815, -2.613540, -0.777034, 1.570796, 1.706435],accel_mss,speed_ms,0,blend_radius_m)
    |   movel([0.135633, -1.322121, -2.613349, -0.776918, 1.570796, 1.706429],accel_mss,speed_ms,0,blend_radius_m)
    |   movel([0.135314, -1.322429, -2.613157, -0.776803, 1.570796, 1.706110],accel_mss,speed_ms,0,blend_radius_m)
    |   movel([0.135031, -1.322549, -2.613082, -0.776757, 1.570796, 1.705828],accel_mss,speed_ms,0,blend_radius_m)
    |   movel([0.134712, -1.322559, -2.613076, -0.776754, 1.570796, 1.705508],accel_mss,speed_ms,0,blend_radius_m)
    |   movel([0.134730, -1.322156, -2.613328, -0.776906, 1.570796, 1.705526],accel_mss,speed_ms,0,blend_radius_m)
    |   movel([0.134718, -1.321824, -2.613534, -0.777030, 1.570796, 1.705515],accel_mss,speed_ms,0,blend_radius_m)
    |   movel([0.134682, -1.321541, -2.613711, -0.777137, 1.570796, 1.705478],accel_mss,speed_ms,0,blend_radius_m)
    |   movel([0.134613, -1.321296, -2.613863, -0.777229, 1.570796, 1.705410],accel_mss,speed_ms,0,blend_radius_m)
    |   movel([0.134557, -1.321090, -2.613992, -0.777307, 1.570796, 1.705354],accel_mss,speed_ms,0,blend_radius_m)
    |   movel([0.134502, -1.320724, -2.614219, -0.777446, 1.570796, 1.705299],accel_mss,speed_ms,0,blend_radius_m)
    |   movel([0.134451, -1.320298, -2.614484, -0.777607, 1.570796, 1.705248],accel_mss,speed_ms,0,blend_radius_m)
    |   movel([0.134415, -1.319860, -2.614756, -0.777773, 1.570796, 1.705211],accel_mss,speed_ms,0,blend_radius_m)
    |   movel([0.134367, -1.319390, -2.615047, -0.777951, 1.570796, 1.705164],accel_mss,speed_ms,0,blend_radius_m)
    |   movel([0.134277, -1.318861, -2.615375, -0.778153, 1.570796, 1.705074],accel_mss,speed_ms,0,blend_radius_m)
    |   movel([0.134162, -1.318360, -2.615685, -0.778344, 1.570796, 1.704959],accel_mss,speed_ms,0,blend_radius_m)
    |   movel([0.134041, -1.317968, -2.615928, -0.778493, 1.570796, 1.704837],accel_mss,speed_ms,0,blend_radius_m)
    |   speed_ms = 0.003
    |   movel([0.134041, -1.304285, -2.609494, -0.798609, 1.570796, 1.704837],accel_mss,speed_ms,0,blend_radius_m)
    |   speed_ms = 1.000
    |   movel([0.134041, -1.278189, -2.596239, -0.837961, 1.570796, 1.704837],accel_mss,speed_ms,0,blend_radius_m)
    |   movel([0.134679, -1.283341, -2.593214, -0.835834, 1.570796, 1.705475],accel_mss,speed_ms,0,blend_radius_m)
    |   movel([0.134679, -1.309362, -2.606402, -0.796625, 1.570796, 1.705475],accel_mss,speed_ms,0,blend_radius_m)
    |   speed_ms = 0.003
    |   movel([0.134679, -1.319550, -2.611214, -0.781625, 1.570796, 1.705475],accel_mss,speed_ms,0,blend_radius_m)
    |   speed_ms = 0.007
    |   movel([0.134980, -1.319504, -2.611243, -0.781642, 1.570796, 1.705777],accel_mss,speed_ms,0,blend_radius_m)
    |   movel([0.135074, -1.319751, -2.611089, -0.781549, 1.570796, 1.705870],accel_mss,speed_ms,0,blend_radius_m)
    |   movel([0.134842, -1.320061, -2.610896, -0.781432, 1.570796, 1.705638],accel_mss,speed_ms,0,blend_radius_m)
    |   movel([0.134566, -1.320480, -2.610635, -0.781273, 1.570796, 1.705362],accel_mss,speed_ms,0,blend_radius_m)
    |   movel([0.134182, -1.321204, -2.610184, -0.781001, 1.570796, 1.704979],accel_mss,speed_ms,0,blend_radius_m)
    |   movel([0.133839, -1.321923, -2.609735, -0.780731, 1.570796, 1.704635],accel_mss,speed_ms,0,blend_radius_m)
    |   movel([0.133730, -1.322271, -2.609518, -0.780600, 1.570796, 1.704526],accel_mss,speed_ms,0,blend_radius_m)
    |   movel([0.133502, -1.322511, -2.609368, -0.780510, 1.570796, 1.704298],accel_mss,speed_ms,0,blend_radius_m)
    |   movel([0.133427, -1.321682, -2.609886, -0.780821, 1.570796, 1.704224],accel_mss,speed_ms,0,blend_radius_m)
    |   movel([0.133590, -1.320888, -2.610381, -0.781120, 1.570796, 1.704386],accel_mss,speed_ms,0,blend_radius_m)
    |   movel([0.133827, -1.320304, -2.610745, -0.781340, 1.570796, 1.704623],accel_mss,speed_ms,0,blend_radius_m)
    |   movel([0.134055, -1.319981, -2.610946, -0.781462, 1.570796, 1.704851],accel_mss,speed_ms,0,blend_radius_m)
    |   movel([0.134353, -1.319717, -2.611110, -0.781561, 1.570796, 1.705150],accel_mss,speed_ms,0,blend_radius_m)
    |   movel([0.134679, -1.319550, -2.611214, -0.781625, 1.570796, 1.705475],accel_mss,speed_ms,0,blend_radius_m)
    |   speed_ms = 0.003
    |   movel([0.134679, -1.322999, -2.612801, -0.776589, 1.570796, 1.705475],accel_mss,speed_ms,0,blend_radius_m)
    |   speed_ms = 0.007
    |   movel([0.134980, -1.322953, -2.612830, -0.776606, 1.570796, 1.705777],accel_mss,speed_ms,0,blend_radius_m)
    |   movel([0.135074, -1.323199, -2.612676, -0.776514, 1.570796, 1.705870],accel_mss,speed_ms,0,blend_radius_m)
    |   movel([0.134842, -1.323509, -2.612483, -0.776397, 1.570796, 1.705638],accel_mss,speed_ms,0,blend_radius_m)
    |   movel([0.134566, -1.323927, -2.612221, -0.776241, 1.570796, 1.705362],accel_mss,speed_ms,0,blend_radius_m)
    |   movel([0.134182, -1.324649, -2.611769, -0.775971, 1.570796, 1.704979],accel_mss,speed_ms,0,blend_radius_m)
    |   movel([0.133839, -1.325366, -2.611319, -0.775704, 1.570796, 1.704635],accel_mss,speed_ms,0,blend_radius_m)
    |   movel([0.133730, -1.325714, -2.611100, -0.775575, 1.570796, 1.704526],accel_mss,speed_ms,0,blend_radius_m)
    |   movel([0.133502, -1.325953, -2.610950, -0.775486, 1.570796, 1.704298],accel_mss,speed_ms,0,blend_radius_m)
    |   movel([0.133427, -1.325126, -2.611469, -0.775794, 1.570796, 1.704224],accel_mss,speed_ms,0,blend_radius_m)
    |   movel([0.133590, -1.324334, -2.611966, -0.776089, 1.570796, 1.704386],accel_mss,speed_ms,0,blend_radius_m)
    |   movel([0.133827, -1.323751, -2.612331, -0.776307, 1.570796, 1.704623],accel_mss,speed_ms,0,blend_radius_m)
    |   movel([0.134055, -1.323428, -2.612533, -0.776428, 1.570796, 1.704851],accel_mss,speed_ms,0,blend_radius_m)
    |   movel([0.134353, -1.323166, -2.612697, -0.776526, 1.570796, 1.705150],accel_mss,speed_ms,0,blend_radius_m)
    |   movel([0.134679, -1.322999, -2.612801, -0.776589, 1.570796, 1.705475],accel_mss,speed_ms,0,blend_radius_m)
    |   speed_ms = 0.003
    |   movel([0.134679, -1.309362, -2.606402, -0.796625, 1.570796, 1.705475],accel_mss,speed_ms,0,blend_radius_m)
    |   speed_ms = 1.000
    |   movel([0.134679, -1.283341, -2.593214, -0.835834, 1.570796, 1.705475],accel_mss,speed_ms,0,blend_radius_m)
    |   movel([0.131149, -1.284706, -2.592407, -0.835275, 1.570796, 1.701945],accel_mss,speed_ms,0,blend_radius_m)
    |   movel([0.131149, -1.310707, -2.605577, -0.796105, 1.570796, 1.701945],accel_mss,speed_ms,0,blend_radius_m)
    |   speed_ms = 0.003
    |   movel([0.131149, -1.320886, -2.610383, -0.781120, 1.570796, 1.701945],accel_mss,speed_ms,0,blend_radius_m)
    |   speed_ms = 0.007
    |   movel([0.131120, -1.321932, -2.609730, -0.780727, 1.570796, 1.701916],accel_mss,speed_ms,0,blend_radius_m)
    |   movel([0.131035, -1.323492, -2.608753, -0.780143, 1.570796, 1.701832],accel_mss,speed_ms,0,blend_radius_m)
    |   movel([0.131017, -1.323858, -2.608524, -0.780007, 1.570796, 1.701813],accel_mss,speed_ms,0,blend_radius_m)
    |   movel([0.130997, -1.324146, -2.608344, -0.779900, 1.570796, 1.701794],accel_mss,speed_ms,0,blend_radius_m)
    |   movel([0.130123, -1.324846, -2.607904, -0.779639, 1.570796, 1.700920],accel_mss,speed_ms,0,blend_radius_m)
    |   movel([0.128228, -1.325645, -2.607401, -0.779343, 1.570796, 1.699025],accel_mss,speed_ms,0,blend_radius_m)
    |   movel([0.125807, -1.326573, -2.606816, -0.779000, 1.570796, 1.696603],accel_mss,speed_ms,0,blend_radius_m)
    |   movel([0.122872, -1.327600, -2.606167, -0.778622, 1.570796, 1.693668],accel_mss,speed_ms,0,blend_radius_m)
    |   movel([0.119571, -1.328664, -2.605494, -0.778231, 1.570796, 1.690367],accel_mss,speed_ms,0,blend_radius_m)
    |   movel([0.115001, -1.330030, -2.604627, -0.777732, 1.570796, 1.685797],accel_mss,speed_ms,0,blend_radius_m)
    |   movel([0.110560, -1.331316, -2.603808, -0.777265, 1.570796, 1.681356],accel_mss,speed_ms,0,blend_radius_m)
    |   movel([0.108416, -1.331838, -2.603475, -0.777076, 1.570796, 1.679213],accel_mss,speed_ms,0,blend_radius_m)
    |   movel([0.106983, -1.332105, -2.603304, -0.776979, 1.570796, 1.677779],accel_mss,speed_ms,0,blend_radius_m)
    |   movel([0.105904, -1.332248, -2.603213, -0.776927, 1.570796, 1.676701],accel_mss,speed_ms,0,blend_radius_m)
    |   movel([0.105130, -1.332283, -2.603191, -0.776915, 1.570796, 1.675926],accel_mss,speed_ms,0,blend_radius_m)
    |   movel([0.104723, -1.332186, -2.603253, -0.776950, 1.570796, 1.675519],accel_mss,speed_ms,0,blend_radius_m)
    |   movel([0.104426, -1.332017, -2.603361, -0.777011, 1.570796, 1.675223],accel_mss,speed_ms,0,blend_radius_m)
    |   movel([0.104710, -1.330110, -2.604576, -0.777703, 1.570796, 1.675506],accel_mss,speed_ms,0,blend_radius_m)
    |   movel([0.104834, -1.329350, -2.605059, -0.777981, 1.570796, 1.675631],accel_mss,speed_ms,0,blend_radius_m)
    |   movel([0.104958, -1.328701, -2.605470, -0.778218, 1.570796, 1.675754],accel_mss,speed_ms,0,blend_radius_m)
    |   movel([0.105079, -1.328161, -2.605812, -0.778416, 1.570796, 1.675875],accel_mss,speed_ms,0,blend_radius_m)
    |   movel([0.105303, -1.327938, -2.605954, -0.778498, 1.570796, 1.676100],accel_mss,speed_ms,0,blend_radius_m)
    |   movel([0.105929, -1.327746, -2.606075, -0.778568, 1.570796, 1.676725],accel_mss,speed_ms,0,blend_radius_m)
    |   movel([0.106794, -1.327508, -2.606225, -0.778656, 1.570796, 1.677590],accel_mss,speed_ms,0,blend_radius_m)
    |   movel([0.108053, -1.327188, -2.606428, -0.778773, 1.570796, 1.678850],accel_mss,speed_ms,0,blend_radius_m)
    |   movel([0.112633, -1.325957, -2.607204, -0.779228, 1.570796, 1.683429],accel_mss,speed_ms,0,blend_radius_m)
    |   movel([0.118191, -1.324293, -2.608251, -0.779845, 1.570796, 1.688988],accel_mss,speed_ms,0,blend_radius_m)
    |   movel([0.123775, -1.322501, -2.609374, -0.780514, 1.570796, 1.694571],accel_mss,speed_ms,0,blend_radius_m)
    |   movel([0.128427, -1.320864, -2.610396, -0.781129, 1.570796, 1.699223],accel_mss,speed_ms,0,blend_radius_m)
    |   movel([0.129521, -1.320464, -2.610645, -0.781279, 1.570796, 1.700318],accel_mss,speed_ms,0,blend_radius_m)
    |   movel([0.130326, -1.320191, -2.610816, -0.781383, 1.570796, 1.701122],accel_mss,speed_ms,0,blend_radius_m)
    |   movel([0.130928, -1.320001, -2.610934, -0.781454, 1.570796, 1.701725],accel_mss,speed_ms,0,blend_radius_m)
    |   movel([0.131147, -1.320138, -2.610849, -0.781403, 1.570796, 1.701943],accel_mss,speed_ms,0,blend_radius_m)
    |   movel([0.131149, -1.320886, -2.610383, -0.781120, 1.570796, 1.701945],accel_mss,speed_ms,0,blend_radius_m)
    |   speed_ms = 0.003
    |   movel([0.131149, -1.324332, -2.611968, -0.776090, 1.570796, 1.701945],accel_mss,speed_ms,0,blend_radius_m)
    |   speed_ms = 0.007
    |   movel([0.131120, -1.325375, -2.611313, -0.775701, 1.570796, 1.701916],accel_mss,speed_ms,0,blend_radius_m)
    |   movel([0.131035, -1.326932, -2.610334, -0.775123, 1.570796, 1.701832],accel_mss,speed_ms,0,blend_radius_m)
    |   movel([0.131017, -1.327296, -2.610104, -0.774989, 1.570796, 1.701813],accel_mss,speed_ms,0,blend_radius_m)
    |   movel([0.130997, -1.327583, -2.609923, -0.774882, 1.570796, 1.701794],accel_mss,speed_ms,0,blend_radius_m)
    |   movel([0.130123, -1.328282, -2.609482, -0.774625, 1.570796, 1.700920],accel_mss,speed_ms,0,blend_radius_m)
    |   movel([0.128228, -1.329079, -2.608978, -0.774332, 1.570796, 1.699025],accel_mss,speed_ms,0,blend_radius_m)
    |   movel([0.125807, -1.330005, -2.608391, -0.773993, 1.570796, 1.696603],accel_mss,speed_ms,0,blend_radius_m)
    |   movel([0.122872, -1.331030, -2.607741, -0.773619, 1.570796, 1.693668],accel_mss,speed_ms,0,blend_radius_m)
    |   movel([0.119571, -1.332091, -2.607065, -0.773233, 1.570796, 1.690367],accel_mss,speed_ms,0,blend_radius_m)
    |   movel([0.115001, -1.333453, -2.606196, -0.772739, 1.570796, 1.685797],accel_mss,speed_ms,0,blend_radius_m)
    |   movel([0.110560, -1.334736, -2.605376, -0.772277, 1.570796, 1.681356],accel_mss,speed_ms,0,blend_radius_m)
    |   movel([0.108416, -1.335257, -2.605042, -0.772090, 1.570796, 1.679213],accel_mss,speed_ms,0,blend_radius_m)
    |   movel([0.106983, -1.335524, -2.604871, -0.771995, 1.570796, 1.677779],accel_mss,speed_ms,0,blend_radius_m)
    |   movel([0.105904, -1.335667, -2.604779, -0.771943, 1.570796, 1.676701],accel_mss,speed_ms,0,blend_radius_m)
    |   movel([0.105130, -1.335701, -2.604757, -0.771931, 1.570796, 1.675926],accel_mss,speed_ms,0,blend_radius_m)
    |   movel([0.104723, -1.335604, -2.604819, -0.771966, 1.570796, 1.675519],accel_mss,speed_ms,0,blend_radius_m)
    |   movel([0.104426, -1.335435, -2.604927, -0.772026, 1.570796, 1.675223],accel_mss,speed_ms,0,blend_radius_m)
    |   movel([0.104710, -1.333533, -2.606145, -0.772710, 1.570796, 1.675506],accel_mss,speed_ms,0,blend_radius_m)
    |   movel([0.104834, -1.332775, -2.606630, -0.772985, 1.570796, 1.675631],accel_mss,speed_ms,0,blend_radius_m)
    |   movel([0.104958, -1.332128, -2.607042, -0.773219, 1.570796, 1.675754],accel_mss,speed_ms,0,blend_radius_m)
    |   movel([0.105079, -1.331589, -2.607385, -0.773415, 1.570796, 1.675875],accel_mss,speed_ms,0,blend_radius_m)
    |   movel([0.105303, -1.331366, -2.607527, -0.773496, 1.570796, 1.676100],accel_mss,speed_ms,0,blend_radius_m)
    |   movel([0.105929, -1.331175, -2.607648, -0.773565, 1.570796, 1.676725],accel_mss,speed_ms,0,blend_radius_m)
    |   movel([0.106794, -1.330938, -2.607799, -0.773652, 1.570796, 1.677590],accel_mss,speed_ms,0,blend_radius_m)
    |   movel([0.108053, -1.330618, -2.608002, -0.773769, 1.570796, 1.678850],accel_mss,speed_ms,0,blend_radius_m)
    |   movel([0.112633, -1.329391, -2.608781, -0.774218, 1.570796, 1.683429],accel_mss,speed_ms,0,blend_radius_m)
    |   movel([0.118191, -1.327730, -2.609830, -0.774828, 1.570796, 1.688988],accel_mss,speed_ms,0,blend_radius_m)
    |   movel([0.123775, -1.325943, -2.610956, -0.775490, 1.570796, 1.694571],accel_mss,speed_ms,0,blend_radius_m)
    |   movel([0.128427, -1.324310, -2.611981, -0.776098, 1.570796, 1.699223],accel_mss,speed_ms,0,blend_radius_m)
    |   movel([0.129521, -1.323911, -2.612231, -0.776247, 1.570796, 1.700318],accel_mss,speed_ms,0,blend_radius_m)
    |   movel([0.130326, -1.323638, -2.612402, -0.776349, 1.570796, 1.701122],accel_mss,speed_ms,0,blend_radius_m)
    |   movel([0.130928, -1.323448, -2.612520, -0.776420, 1.570796, 1.701725],accel_mss,speed_ms,0,blend_radius_m)
    |   movel([0.131147, -1.323585, -2.612435, -0.776369, 1.570796, 1.701943],accel_mss,speed_ms,0,blend_radius_m)
    |   movel([0.131149, -1.324332, -2.611968, -0.776090, 1.570796, 1.701945],accel_mss,speed_ms,0,blend_radius_m)
    |   speed_ms = 0.003
    |   movel([0.131149, -1.310707, -2.605577, -0.796105, 1.570796, 1.701945],accel_mss,speed_ms,0,blend_radius_m)
    |   speed_ms = 1.000
    |   movel([0.131149, -1.284706, -2.592407, -0.835275, 1.570796, 1.701945],accel_mss,speed_ms,0,blend_radius_m)
    |   movel([0.130246, -1.289093, -2.589799, -0.833497, 1.570796, 1.701042],accel_mss,speed_ms,0,blend_radius_m)
    |   movel([0.130246, -1.315028, -2.602912, -0.794450, 1.570796, 1.701042],accel_mss,speed_ms,0,blend_radius_m)
    |   speed_ms = 0.003
    |   movel([0.130246, -1.325177, -2.607695, -0.779516, 1.570796, 1.701042],accel_mss,speed_ms,0,blend_radius_m)
    |   speed_ms = 0.007
    |   movel([0.130537, -1.325159, -2.607707, -0.779523, 1.570796, 1.701333],accel_mss,speed_ms,0,blend_radius_m)
    |   movel([0.130658, -1.325582, -2.607441, -0.779367, 1.570796, 1.701454],accel_mss,speed_ms,0,blend_radius_m)
    |   movel([0.130573, -1.325899, -2.607241, -0.779249, 1.570796, 1.701369],accel_mss,speed_ms,0,blend_radius_m)
    |   movel([0.128623, -1.326507, -2.606858, -0.779025, 1.570796, 1.699420],accel_mss,speed_ms,0,blend_radius_m)
    |   movel([0.127749, -1.326789, -2.606680, -0.778921, 1.570796, 1.698546],accel_mss,speed_ms,0,blend_radius_m)
    |   movel([0.127105, -1.327017, -2.606536, -0.778836, 1.570796, 1.697901],accel_mss,speed_ms,0,blend_radius_m)
    |   movel([0.126634, -1.327205, -2.606417, -0.778767, 1.570796, 1.697431],accel_mss,speed_ms,0,blend_radius_m)
    |   movel([0.126266, -1.327534, -2.606209, -0.778646, 1.570796, 1.697062],accel_mss,speed_ms,0,blend_radius_m)
    |   movel([0.126079, -1.327830, -2.606022, -0.778537, 1.570796, 1.696875],accel_mss,speed_ms,0,blend_radius_m)
    |   movel([0.125897, -1.328192, -2.605793, -0.778404, 1.570796, 1.696694],accel_mss,speed_ms,0,blend_radius_m)
    |   movel([0.125732, -1.328601, -2.605534, -0.778255, 1.570796, 1.696528],accel_mss,speed_ms,0,blend_radius_m)
    |   movel([0.125552, -1.328903, -2.605342, -0.778144, 1.570796, 1.696348],accel_mss,speed_ms,0,blend_radius_m)
    |   movel([0.125246, -1.329124, -2.605202, -0.778063, 1.570796, 1.696042],accel_mss,speed_ms,0,blend_radius_m)
    |   movel([0.124966, -1.329233, -2.605133, -0.778023, 1.570796, 1.695762],accel_mss,speed_ms,0,blend_radius_m)
    |   movel([0.122675, -1.329915, -2.604700, -0.777774, 1.570796, 1.693471],accel_mss,speed_ms,0,blend_radius_m)
    |   movel([0.120052, -1.330689, -2.604208, -0.777493, 1.570796, 1.690849],accel_mss,speed_ms,0,blend_radius_m)
    |   movel([0.117013, -1.331578, -2.603641, -0.777170, 1.570796, 1.687809],accel_mss,speed_ms,0,blend_radius_m)
    |   movel([0.109157, -1.333892, -2.602162, -0.776335, 1.570796, 1.679954],accel_mss,speed_ms,0,blend_radius_m)
    |   movel([0.108940, -1.333692, -2.602290, -0.776407, 1.570796, 1.679737],accel_mss,speed_ms,0,blend_radius_m)
    |   movel([0.108795, -1.333473, -2.602430, -0.776486, 1.570796, 1.679591],accel_mss,speed_ms,0,blend_radius_m)
    |   movel([0.108753, -1.333230, -2.602586, -0.776573, 1.570796, 1.679550],accel_mss,speed_ms,0,blend_radius_m)
    |   movel([0.108706, -1.332977, -2.602748, -0.776664, 1.570796, 1.679502],accel_mss,speed_ms,0,blend_radius_m)
    |   movel([0.108544, -1.332738, -2.602900, -0.776751, 1.570796, 1.679341],accel_mss,speed_ms,0,blend_radius_m)
    |   movel([0.108405, -1.332544, -2.603025, -0.776821, 1.570796, 1.679202],accel_mss,speed_ms,0,blend_radius_m)
    |   movel([0.110094, -1.331856, -2.603464, -0.777069, 1.570796, 1.680890],accel_mss,speed_ms,0,blend_radius_m)
    |   movel([0.111895, -1.331317, -2.603808, -0.777265, 1.570796, 1.682692],accel_mss,speed_ms,0,blend_radius_m)
    |   movel([0.114019, -1.330699, -2.604201, -0.777489, 1.570796, 1.684815],accel_mss,speed_ms,0,blend_radius_m)
    |   movel([0.119034, -1.329206, -2.605150, -0.778033, 1.570796, 1.689830],accel_mss,speed_ms,0,blend_radius_m)
